	MotorRunning			: ARRAY[1..6] OF BOOL;
	
	AutoMode				: BOOL;
	
	VibrationSensorX		: ARRAY[1..6] OF REAL;
	VibrationSensorY		: ARRAY[1..6] OF REAL;
	VibrationSensorZ 		: ARRAY[1..6] OF REAL;
	VibrationSensorsEnable	: BOOL := TRUE;
	
	AirFlowRate				: REAL;
	AirPressure				: REAL;
	AirTemperature			: REAL;
	
	AirValve				: ARRAY[1..6] OF AirValveSimSignals;
	AirValveEnable			: ARRAY[1..6] OF BOOL := [TRUE, TRUE, TRUE, TRUE];
	AirValvePositionSim		: ARRAY [1..6] OF INT;
	
	ProductPosition			: INT;
	SensorProductActive		: BOOL;	
	OkProductCount			: UINT;
	NokProductCount			: UINT;	
	OkPartsPerMinRate		: UINT;	
	OkPartsPerMinHistorical	: ARRAY [1..5] OF INT;
	
	ElCurrentL1				: ARRAY[1..2] OF REAL;
	ElCurrentL2				: ARRAY[1..2] OF REAL;
	ElCurrentL3				: ARRAY[1..2] OF REAL;
	
	AmbientTemperature		: REAL;
	AmbientHumidity			: REAL;
	
	OilDiffPressure			: REAL;
	
END_VAR

// ---- POUs/PRG_10ms/PRG_01_MAIN.TcPOU
PROGRAM PRG_01_MAIN
VAR
			tonRecycle100ms			:	TON;
			tonRecycle5sec			:	TON;
END_VAR

PRG_02_DataMapping();

Simulation();

PRG_03_VibrationAnalytics();
PRG_04_AirValveAnalytics();
PRG_05_ElectricalAnalytics();
PRG_06_ElectricalMonitoring();
PRG_07_LineState();
PRG_08_ProductionStatistics();
PRG_09_PlcDiagnostic();


tonRecycle5sec(IN:=NOT tonRecycle5sec.Q, PT:=T#5S);
tonRecycle100ms(IN:=NOT tonRecycle100ms.Q, PT:=T#500MS);

// 500 ms cycle monitoring
IF tonRecycle100ms.Q THEN
	PRG_11_AirFlowAnalytics();
	
END_IF

// slow process values monitoring
IF tonRecycle5sec.Q THEN
	PRG_10_TempHumidAnalytics();
	PRG_12_OilContaminationAnalytics();
END_IF

END_PROGRAM

// ---- POUs/PRG_10ms/PRG_02_DataMapping.TcPOU
PROGRAM PRG_02_DataMapping
VAR

END_VAR


// ************** IO-Link node 1 ***************
GVL_SW.VibSensor1AccelRmsX 	:= GVL_HW.IoLinkNode1Ch1_VibAccelRmsX;
GVL_SW.VibSensor1AccelRmsY 	:= GVL_HW.IoLinkNode1Ch1_VibAccelRmsY;
GVL_SW.VibSensor1AccelRmsZ 	:= GVL_HW.IoLinkNode1Ch1_VibAccelRmsZ;
GVL_SW.VibSensor1Temp 		:= GVL_HW.IoLinkNode1Ch1_SensorTemp;

GVL_SW.VibSensor2AccelRmsX 	:= GVL_HW.IoLinkNode1Ch2_VibAccelRmsX;
GVL_SW.VibSensor2AccelRmsY 	:= GVL_HW.IoLinkNode1Ch2_VibAccelRmsY;
GVL_SW.VibSensor2AccelRmsZ 	:= GVL_HW.IoLinkNode1Ch2_VibAccelRmsZ;
GVL_SW.VibSensor2Temp 		:= GVL_HW.IoLinkNode1Ch2_SensorTemp;

GVL_SW.VibSensor3AccelRmsX 	:= GVL_HW.IoLinkNode1Ch3_VibAccelRmsX;
GVL_SW.VibSensor3AccelRmsY 	:= GVL_HW.IoLinkNode1Ch3_VibAccelRmsY;
GVL_SW.VibSensor3AccelRmsZ 	:= GVL_HW.IoLinkNode1Ch3_VibAccelRmsZ;
GVL_SW.VibSensor3Temp 		:= GVL_HW.IoLinkNode1Ch3_SensorTemp;

GVL_SW.VibSensor4AccelRmsX 	:= GVL_HW.IoLinkNode1Ch4_VibAccelRmsX;
GVL_SW.VibSensor4AccelRmsY 	:= GVL_HW.IoLinkNode1Ch4_VibAccelRmsY;
GVL_SW.VibSensor4AccelRmsZ 	:= GVL_HW.IoLinkNode1Ch4_VibAccelRmsZ;
GVL_SW.VibSensor4Temp 		:= GVL_HW.IoLinkNode1Ch4_SensorTemp;

GVL_SW.VibSensor5AccelRmsX 	:= GVL_HW.IoLinkNode1Ch5_VibAccelRmsX;
GVL_SW.VibSensor5AccelRmsY 	:= GVL_HW.IoLinkNode1Ch5_VibAccelRmsY;
GVL_SW.VibSensor5AccelRmsZ 	:= GVL_HW.IoLinkNode1Ch5_VibAccelRmsZ;
GVL_SW.VibSensor5Temp 		:= GVL_HW.IoLinkNode1Ch5_SensorTemp;

GVL_SW.VibSensor6AccelRmsX 	:= GVL_HW.IoLinkNode1Ch6_VibAccelRmsX;
GVL_SW.VibSensor6AccelRmsY 	:= GVL_HW.IoLinkNode1Ch6_VibAccelRmsY;
GVL_SW.VibSensor6AccelRmsZ 	:= GVL_HW.IoLinkNode1Ch6_VibAccelRmsZ;
GVL_SW.VibSensor6Temp 		:= GVL_HW.IoLinkNode1Ch6_SensorTemp;


// ************** IO-Link node 2 ***************
GVL_SW.AirMassFlowRate		:= GVL_HW.IoLinkNode2Ch1_MassFlowRate;	
GVL_SW.AirFlowVelocity		:= GVL_HW.IoLinkNode2Ch1_FlowVelocity;
GVL_SW.AirVolume			:= GVL_HW.IoLinkNode2Ch1_Volume;
GVL_SW.AirVolumetricFlowRate := (GVL_HW.IoLinkNode2Ch1_VolFlowRate * 1000) / 60.0;		// convert [m3/h] to [l/min]
GVL_SW.AirMass				:= GVL_HW.IoLinkNode2Ch1_Mass;
GVL_SW.AirEnergy			:= GVL_HW.IoLinkNode2Ch1_Energy;
GVL_SW.AirTemperature		:= GVL_HW.IoLinkNode2Ch1_Temperature;
GVL_SW.AirPressure			:= GVL_HW.IoLinkNode2Ch1_Pressure;

GVL_SW.AmbientTempSensor 	:=  UINT_TO_REAL( SHL(GVL_HW.IoLinkNode2Ch2_Temperature[1], 8) +  
												GVL_HW.IoLinkNode2Ch2_Temperature[2]) / 10.0;
												
GVL_SW.AmbientHumiditySensor :=  UINT_TO_REAL(SHL(GVL_HW.IoLinkNode2Ch2_Humidity[1], 8) + 
													GVL_HW.IoLinkNode2Ch2_Humidity[1] ) / 10.0;
													
													
GVL_SW.LevelSensor			:=	TO_REAL(GVL_HW.IoLinkNode2Ch3_Level) / 1000.0;			// convert to m with 1mm resolution
GVL_SW.DiffPressSensor		:= 	TO_REAL(GVL_HW.IoLinkNode2Ch4_DiffPress) / 10;			// convert to bar with 0.1 bar resolution

// Profinet IO-device data
GVL_SW.PnIoDevice_32Word_In 	:= GVL_HW.PnIoDevice_32Word_In;
GVL_SW.PnIoDevice_32DWord_In 	:= GVL_HW.PnIoDevice_32DWord_In;
GVL_SW.PnIoDevice_10Real_In		:= GVL_HW.PnIoDevice_10Real_In;
GVL_SW.PnIoDevice_10Real_Out	:= GVL_HW.PnIoDevice_10Real_Out;

// Here it's place for specified mapping of GVL_SW.PnIoDevice e.g.
// GVL_SW.Motor1.SignalStart :=  GVL_HW.PnIoDevice_32Word_In[1].0;
// GVL_SW.AnalogValue1 := GVL_HW.PnIoDevice_10Real_In[0].1;

END_PROGRAM

// ---- POUs/PRG_10ms/Simulation.TcPOU
PROGRAM Simulation
VAR
	idx			: BYTE;
	tp1Motor 	: ARRAY[1..6] OF TP;
	tp2Motor 	: ARRAY[1..6] OF TP;
	
	VibSensorBase : ARRAY[1..6] OF REAL := [0.7, 0.2, 0.3, 0.8, 0.5, 0.1];
	VibSensorOffset : ARRAY[1..6] OF REAL;
	
	AirFlowRateBase			:	REAL := 30.0;
	AirPressureBase			:	REAL := 6.0;
	AirTemperatureBase		:	REAL := 20.0;
	
	AirValve				:	ARRAY [1..6] OF Valve_Signal_Sim;
	AirValvePositionSim		: 	ARRAY [1..6] OF INT;
	
	tonProductPos			:	TON;
	rtrigProductSensor		: 	R_TRIG;
	
	tp1AutoMode				:	TP;
	tp2AutoMode				:	TP;
	tp1AutoModeTime			:	TIME := T#5S;
	tp2AutoModeTime			:	TIME := T#2S;
	rtrigAutoMode			:	R_TRIG;

	rndTime1				: INT;
	rndTime2				: INT;
	
	ElecSample1				: INT;
	ElecSample2				: INT;
	ElecCurrentOffsetL1		: REAL;
	ElecCurrentOffsetL2		: REAL;	
	ElecCurrentOffsetL3		: REAL;
	ElCurrentL1Base			: ARRAY[1..2] OF ARRAY[1..100] OF REAL := 
								[
								[0, 0, 0.1, 0.3, 0.45, 0.60, 0.70, 0.80, 0.95, 1.1, 1.3, 1.4, 1.55, 1.6, 1.59,1.55, 
								1.45, 1.3, 1.2, 1.1, 1.05, 1.0, 0.95, 0.9, 0.85, 0.83, 0.80, 0.78, 0.75, 0.74, 0.72,
								0.70, 0.69, 0.69, 0.69, 0.68, 0.68, 0.67, 0.67, 0.65, 0.64, 0.62, 0.60, 0.58, 0.58, 0.57, 0.56, 0.55, 0.55,
								0, 0, 0, 0, 0, 0, 0, 0, 0, 0],
								[0, 0, 0.1, 0.2, 0.3, 0.55, 1.0, 1.3, 1.5, 1.7, 1.8, 1.81, 1.7, 1.5, 1.2, 1.22, 1.19, 1.23,
								1.19, 1.21, 1.18, 1.22, 1.19, 1.23, 1.17, 1.21, 1.20, 1.18, 1.21, 1.18, 1.22, 1.17, 1.23,
								1.19, 1.21, 1.19, 1.20, 1.19, 1.20, 1.19, 1.21, 1.20, 1.20, 1.22, 1.19, 1.21, 1.18, 1.21, 1.2, 1.2,
								1.21, 1.20, 1.20, 1.22, 1.19, 1.21, 1.18, 1.21, 1.2, 1.2, 40(1.2)]];
								
	ElCurrentL2Base			: ARRAY[1..2] OF ARRAY[1..100] OF REAL := 
								[
								[0, 0, 0.1, 0.3, 0.45, 0.60, 0.70, 0.80, 0.95, 1.1, 1.3, 1.4, 1.55, 1.6, 1.59,1.55, 
								1.45, 1.3, 1.2, 1.1, 1.05, 1.0, 0.95, 0.9, 0.85, 0.83, 0.80, 0.78, 0.75, 0.74, 0.72,
								0.70, 0.69, 0.69, 0.69, 0.68, 0.68, 0.67, 0.67, 0.65, 0.64, 0.62, 0.60, 0.58, 0.58, 0.57, 0.56, 0.55, 0.55,
								0, 0, 0, 0, 0, 0, 0, 0, 0, 0],
								[0, 0, 0.1, 0.2, 0.3, 0.55, 1.0, 1.3, 1.5, 1.7, 1.8, 1.81, 1.7, 1.5, 1.2, 1.22, 1.19, 1.23,
								1.19, 1.21, 1.18, 1.22, 1.19, 1.23, 1.17, 1.21, 1.20, 1.18, 1.21, 1.18, 1.22, 1.17, 1.23,
								1.19, 1.21, 1.19, 1.20, 1.19, 1.20, 1.19, 1.21, 1.20, 1.20, 1.22, 1.19, 1.21, 1.18, 1.21, 1.2, 1.2,
								1.21, 1.20, 1.20, 1.22, 1.19, 1.21, 1.18, 1.21, 1.2, 1.2]];

	ElCurrentL3Base			: ARRAY[1..2] OF ARRAY[1..100] OF REAL := 
								[
								[0, 0, 0.1, 0.3, 0.45, 0.60, 0.70, 0.80, 0.95, 1.1, 1.3, 1.4, 1.55, 1.6, 1.59,1.55, 
								1.45, 1.3, 1.2, 1.1, 1.05, 1.0, 0.95, 0.9, 0.85, 0.83, 0.80, 0.78, 0.75, 0.74, 0.72,
								0.70, 0.69, 0.69, 0.69, 0.68, 0.68, 0.67, 0.67, 0.65, 0.64, 0.62, 0.60, 0.58, 0.58, 0.57, 0.56, 0.55, 0.55,
								0, 0, 0, 0, 0, 0, 0, 0, 0, 0],
								[0, 0, 0.1, 0.2, 0.3, 0.55, 1.0, 1.3, 1.5, 1.7, 1.8, 1.81, 1.7, 1.5, 1.2, 1.22, 1.19, 1.23,
								1.19, 1.21, 1.18, 1.22, 1.19, 1.23, 1.17, 1.21, 1.20, 1.18, 1.21, 1.18, 1.22, 1.17, 1.23,
								1.19, 1.21, 1.19, 1.20, 1.19, 1.20, 1.19, 1.21, 1.20, 1.20, 1.22, 1.19, 1.21, 1.18, 1.21, 1.2, 1.2,
								1.21, 1.20, 1.20, 1.22, 1.19, 1.21, 1.18, 1.21, 1.2, 1.2]];
END_VAR

IF GVL_Visu.ButtonStart THEN
	
	GVL_Visu.LineRunning := TRUE;
	// simulate motor running signals
	tp1Motor[1](IN:= NOT tp2Motor[1].Q, PT:= T#1S);
	tp2Motor[1](IN:= NOT tp1Motor[1].Q, PT:= T#500MS);
	
	tp1Motor[2](IN:= NOT tp2Motor[2].Q, PT:= T#2S);
	tp2Motor[2](IN:= NOT tp1Motor[2].Q, PT:= T#300MS);
	
	tp1Motor[3](IN:= NOT tp2Motor[3].Q, PT:= T#1.7S);
	tp2Motor[3](IN:= NOT tp1Motor[3].Q, PT:= T#500MS);
	
	tp1Motor[4](IN:= NOT tp2Motor[4].Q, PT:= T#1S);
	tp2Motor[4](IN:= NOT tp1Motor[4].Q, PT:= T#1S);
	
	tp1Motor[5](IN:= NOT tp2Motor[5].Q, PT:= T#500MS);
	tp2Motor[5](IN:= NOT tp1Motor[5].Q, PT:= T#2S);
	
	tp1Motor[6](IN:= NOT tp2Motor[6].Q, PT:= T#1S);
	tp2Motor[6](IN:= NOT tp1Motor[6].Q, PT:= T#300MS);
	
	// simulate auto/manual mode
	tp1AutoMode(IN:= NOT tp2AutoMode.Q, PT:= tp1AutoModeTime);
	tp2AutoMode(IN:= NOT tp1AutoMode.Q, PT:= tp2AutoModeTime);
	
	rtrigAutoMode(CLK:=tp1AutoMode.Q);
	
	// generate random time windows of auto and manual period  
	IF  rtrigAutoMode.Q THEN
		rndTime1 := RDM2(last:=2, low:=0, high:=70);
		tp1AutoModeTime:=T#5S + INT_TO_TIME(rndTime1*100);
		
		rndTime2 := RDM2(last:=5, low:=0, high:=30);
		tp2AutoModeTime:=T#2S + INT_TO_TIME(rndTime2*100);
	END_IF

	GVL_Visu.AutoMode := tp2AutoMode.Q;
	
	
	// simulate vibration sensors
	FOR idx := 1 TO 6 DO
		GVL_Visu.MotorRunning[idx] := tp1Motor[idx].Q;
		
		GVL_Visu.VibrationSensorX[idx] := VibSensorBase[idx] + RDM(0.4);
		GVL_Visu.VibrationSensorY[idx] := VibSensorBase[idx] + RDM(0.2);
		GVL_Visu.VibrationSensorZ[idx] := VibSensorBase[idx] + RDM(0.8);	
	END_FOR
	
	// simulate air supply sensors
	GVL_Visu.AirFlowRate 		:= AirFlowRateBase + 2* RDM(0.5);
	GVL_Visu.AirPressure		:= AirPressureBase + 2 * RDM(0.9); 
	GVL_Visu.AirTemperature		:= AirTemperatureBase + RDM(0.3);
	
	// simulate air valves
	AirValve[1](StartSim			:= TRUE, 
			    ExtendCmdTime		:= T#500MS,
			    ExtendTime 			:= T#1800MS,
			    RetractCmdTime 		:= T#600MS,
			    RetractTime  		:= T#2000MS);
			  
	AirValve[2](StartSim			:= TRUE, 
			    ExtendCmdTime		:= T#50MS,
			    ExtendTime 			:= T#180MS,
			    RetractCmdTime 		:= T#50MS,
			    RetractTime  		:= T#145MS);
				
	AirValve[3](StartSim			:= TRUE, 
			    ExtendCmdTime		:= T#100MS,
			    ExtendTime 			:= T#1200MS,
			    RetractCmdTime 		:= T#120MS,
			    RetractTime  		:= T#1500MS);
				
	AirValve[4](StartSim			:= TRUE, 
			    ExtendCmdTime		:= T#30MS,
			    ExtendTime 			:= T#120MS,
			    RetractCmdTime 		:= T#30MS,
			    RetractTime  		:= T#120MS);
				
	FOR idx := 1 TO 4 DO
		GVL_Visu.AirValve[idx].ExtendCmd := AirValve[idx].ExtendCmd;
		GVL_Visu.AirValve[idx].ExtendFeedback := AirValve[idx].ExtendFeedback;
		GVL_Visu.AirValve[idx].RetractCmd := AirValve[idx].RetractCmd;
		GVL_Visu.AirValve[idx].RetractFeedback := AirValve[idx].RetractFeedback;
		GVL_Visu.AirValvePositionSim[idx] := SEL (NOT GVL_Visu.AirValveEnable[idx], AirValve[idx].nState, 0);
	END_FOR
	
	// simulate product position on the conveyor
	tonProductPos(IN:= NOT tonProductPos.Q, PT:=T#200MS);
	IF tonProductPos.Q THEN
		GVL_Visu.ProductPosition := GVL_Visu.ProductPosition + TO_INT(GVL_Visu.LineSpeed / 5);
	END_IF
	
	IF GVL_Visu.ProductPosition >= 190 THEN
		GVL_Visu.ProductPosition := 0;
	END_IF
	
	// simulate product sensor acitivation
	IF GVL_Visu.ProductPosition >= 175 AND
		 GVL_Visu.ProductPosition <190 THEN
	GVL_Visu.SensorProductActive := TRUE;
	ELSE
		GVL_Visu.SensorProductActive := FALSE;
	END_IF;
	
	// simulate product counting
	rtrigProductSensor(CLK:=GVL_Visu.SensorProductActive);
	IF rtrigProductSensor.Q THEN
		GVL_Visu.OkProductCount := GVL_Visu.OkProductCount + 1;
	END_IF
	
	// simulate electrical current curve of motor 1
	IF GVL_Visu.MotorRunning[1] THEN
		ElecSample1 := ElecSample1+1;
		ElecSample1 := SEL(ElecSample1=60, ElecSample1, 1);
		IF ElecSample1 < 20 OR ElecSample1 > 40 THEN
			ElecCurrentOffsetL1 := RDM(0.67) * 0.05;
			ElecCurrentOffsetL2 := RDM(0.23) * 0.05;
			ElecCurrentOffsetL3 := RDM(0.72) * 0.05;
		ELSE
			ElecCurrentOffsetL1 := RDM(0.31) * 0.05;
			ElecCurrentOffsetL2 := RDM(0.63) * 0.05;
			ElecCurrentOffsetL3 := RDM(0.46) * 0.05;
		END_IF
		GVL_Visu.ElCurrentL1[1] := 	ElCurrentL1Base[1][ElecSample1];
		GVL_Visu.ElCurrentL2[1] := 	ElCurrentL1Base[1][ElecSample1];
		GVL_Visu.ElCurrentL3[1] := 	ElCurrentL1Base[1][ElecSample1];
	ELSE
		ElecSample1 := 0;
		GVL_Visu.ElCurrentL1[1] := 0;
		GVL_Visu.ElCurrentL2[1] := 0;
		GVL_Visu.ElCurrentL3[1] := 0;
	END_IF
	
	// simulate electrical current curve of motor 2
	IF GVL_Visu.MotorRunning[2] THEN
		ElecSample2 := ElecSample2+1;
		ElecSample2 := SEL(ElecSample2=60, ElecSample2, 1);
		GVL_Visu.ElCurrentL1[2] := 	ElCurrentL1Base[2][ElecSample2];
		GVL_Visu.ElCurrentL2[2] := 	ElCurrentL2Base[2][ElecSample2];
		GVL_Visu.ElCurrentL3[2] := 	ElCurrentL3Base[2][ElecSample2];
	ELSE
		ElecSample2 := 0;
		GVL_Visu.ElCurrentL1[2] := 0;
		GVL_Visu.ElCurrentL2[2] := 0;
		GVL_Visu.ElCurrentL3[2] := 0;
	END_IF
	
	// simulate ambient temperature & humidity
	GVL_Visu.AmbientTemperature := 19.0 + 2* RDM(0.7);
	GVL_Visu.AmbientHumidity	:= 60.0 + 3 * RDM(0.5);
	
	// simulate pressure difference for oil contamination sensor
	GVL_Visu.OilDiffPressure := 0.22 + RDM(0.1) * 0.2;
  

ELSE
	GVL_Visu.LineRunning := FALSE;
	tp1AutoMode(IN:=FALSE);
	tp2AutoMode(IN:=FALSE);
	
	GVL_Visu.AutoMode := tp1AutoMode.Q;
	
	FOR idx := 1 TO 4 DO
		AirValve[idx](StartSim := FALSE);
	END_FOR
	
	FOR idx := 1 TO 6 DO
		tp1Motor[idx](IN:= FALSE);
		tp2Motor[idx](IN:= FALSE);	
		GVL_Visu.MotorRunning[idx] := tp1Motor[idx].Q;		
	END_FOR
	
	GVL_Visu.ElCurrentL1[1] := 0;
	GVL_Visu.ElCurrentL2[1] := 0;
	GVL_Visu.ElCurrentL3[1] := 0;
	
	GVL_Visu.ElCurrentL1[2] := 0;
	GVL_Visu.ElCurrentL2[2] := 0;
	GVL_Visu.ElCurrentL3[2] := 0;
	
END_IF

END_PROGRAM

// ---- POUs/FB/Generic/Valve_Signal_Sim.TcPOU
FUNCTION_BLOCK Valve_Signal_Sim
VAR_INPUT
	StartSim : BOOL;
	
	ExtendCmdTime	:	TIME;
	ExtendTime		:	TIME;
	RetractCmdTime	:	TIME;
	RetractTime		:	TIME;
END_VAR
VAR_OUTPUT
	ExtendCmd 		: 	BOOL;
	ExtendFeedback 	: 	BOOL;
	RetractCmd 		: 	BOOL;
	RetractFeedback : 	BOOL;
	SequenceStatus 	: 	INT;
	
END_VAR
VAR
	tonExtendCmd	: TON;
	tonExtend		: TON;
	tonRetractCmd	: TON;
	tonRetract		: TON;
	
	ExtendPos_ton: TON; //czas przebywania na pozycji Extend
	RetractPos_ton: TON; //czas przebywania na pozycji Retract
	
	nState : INT;
	
	// sequence watchdog
	tonWatchdog		: TON;
	rtrigStartSim	: R_TRIG;

	Step20Cnt: INT;
	Step30Cnt: INT;
END_VAR

rtrigStartSim(CLK:=StartSim);

CASE nState OF
0:
	SequenceStatus := 0;
	tonExtendCmd.IN := FALSE;
	tonExtend.IN := FALSE;
	tonRetractCmd.IN := FALSE;
	tonRetract.IN := FALSE;
	
	RetractFeedback := TRUE;
	
	IF rtrigStartSim.Q THEN
		nState := nState + 10;
		tonWatchdog.IN := TRUE;
	END_IF

10:
	SequenceStatus := 10;
	ExtendCmd := TRUE;
	tonExtendCmd.IN := TRUE;
	IF tonExtendCmd.Q THEN
		nState := nState + 10;
		tonExtendCmd.IN := FALSE;
	END_IF
20:	
	SequenceStatus := 20;
	RetractFeedback :=FALSE;
	tonExtend.IN := TRUE;
	IF tonExtend.Q THEN
		nState := nState + 10;
		tonExtend.IN := FALSE;
	END_IF
		
	
30:
	SequenceStatus := 30;
	ExtendFeedback := TRUE;
	ExtendCmd := FALSE;
	ExtendPos_ton.IN := TRUE;
	IF ExtendPos_ton.Q THEN
		nState := nState + 10;
		ExtendPos_ton.IN := FALSE;
	END_IF


40:
	SequenceStatus := 40;
	RetractCmd := TRUE;
	tonRetractCmd.IN := TRUE;
	IF tonRetractCmd.Q THEN
		nState := nState + 10;
		tonRetractCmd.IN := FALSE;
	END_IF
50:
	SequenceStatus := 50;
	ExtendFeedback :=FALSE;
	tonRetract.IN := TRUE;
	IF tonRetract.Q THEN
		nState := nState + 10;
		tonRetract.IN := FALSE;
	END_IF
60:
	SequenceStatus := 60;
	RetractFeedback := TRUE;
	RetractCmd := FALSE;
	RetractPos_ton.IN := TRUE;
	IF RetractPos_ton.Q THEN
		nState := 10;
		RetractPos_ton.IN := FALSE;
	END_IF

	
END_CASE

IF StartSim = FALSE THEN
	nState := 0;
END_IF

tonExtendCmd(PT:=ExtendCmdTime);
tonExtend(PT:=ExtendTime);
tonRetractCmd(PT:=RetractCmdTime);
tonRetract(PT:=RetractTime);

ExtendPos_ton(PT:=T#500MS);
RetractPos_ton(PT:=T#500MS);
tonWatchdog(PT:=T#2H);

END_FUNCTION_BLOCK

// ---- POUs/PRG_10ms/PRG_03_VibrationAnalytics.TcPOU
PROGRAM PRG_03_VibrationAnalytics
VAR
	VibSensor					: ARRAY [1..6] OF VibrationSensor;
	
	
	{attribute 'OPC.UA.DA' := '0'}
	{attribute 'OPC.UA.DA.Access' := '1'}			// read only
	{attribute 'OPC.UA.DA.StructuredType' := '1'}
	VibSensorStruct01			: VibAccelarationDataModel;
	
	{attribute 'OPC.UA.DA' := '0'}
	{attribute 'OPC.UA.DA.Access' := '1'}			// read only
	{attribute 'OPC.UA.DA.StructuredType' := '1'}
	VibSensorStruct02			: VibAccelarationDataModel;

	{attribute 'OPC.UA.DA' := '0'}
	{attribute 'OPC.UA.DA.Access' := '1'}			// read only
	{attribute 'OPC.UA.DA.StructuredType' := '1'}
	VibSensorStruct03			: VibAccelarationDataModel;
	
	{attribute 'OPC.UA.DA' := '0'}
	{attribute 'OPC.UA.DA.Access' := '1'}			// read only
	{attribute 'OPC.UA.DA.StructuredType' := '1'}
	VibSensorStruct04			: VibAccelarationDataModel;
	
	{attribute 'OPC.UA.DA' := '0'}
	{attribute 'OPC.UA.DA.Access' := '1'}			// read only
	{attribute 'OPC.UA.DA.StructuredType' := '1'}
	VibSensorStruct05			: VibAccelarationDataModel;
	
	{attribute 'OPC.UA.DA' := '0'}
	{attribute 'OPC.UA.DA.Access' := '1'}			// read only
	{attribute 'OPC.UA.DA.StructuredType' := '1'}
	VibSensorStruct06			: VibAccelarationDataModel;
	

END_VAR


// PAGE Vibration Sensor 1 ----
VibSensor[1](
    LineName := GVL_const.LineName,
    MachineName := GVL_const.MachineName,
    SensorName := GVL_const.VibSensor1,
    TimeStamp := GVL_SW.Unix_TimeStamp,
    VibAccelX := GVL_Visu.VibrationSensorX[1],
    VibAccelY := GVL_Visu.VibrationSensorY[1],
    VibAccelZ := GVL_Visu.VibrationSensorZ[1],
    SensorTemperature := GVL_SW.VibSensor1Temp,
    MotorState := GVL_Visu.MotorRunning[1],
    Enable := GVL_Visu.LineRunning AND GVL_Visu.VibrationSensorsEnable); // VibrationSensor
VibSensorStruct01 := VibSensor[1].OpcUaVal;

// PAGE Vibration Sensor 2 ---
VibSensor[2](
    LineName := GVL_const.LineName,
    MachineName := GVL_const.MachineName,
    SensorName := GVL_const.VibSensor2,
    TimeStamp := GVL_SW.Unix_TimeStamp,
    VibAccelX := GVL_Visu.VibrationSensorX[2],
    VibAccelY := GVL_Visu.VibrationSensorY[2],
    VibAccelZ := GVL_Visu.VibrationSensorZ[2],
    SensorTemperature := GVL_SW.VibSensor2Temp,
    MotorState := GVL_Visu.MotorRunning[2],
    Enable := GVL_Visu.LineRunning AND GVL_Visu.VibrationSensorsEnable); // VibrationSensor
VibSensorStruct02 := VibSensor[2].OpcUaVal;

// PAGE Vibration Sensor 3 ---
VibSensor[3](
    LineName := GVL_const.LineName,
    MachineName := GVL_const.MachineName,
    SensorName := GVL_const.VibSensor3,
    TimeStamp := GVL_SW.Unix_TimeStamp,
    VibAccelX := GVL_Visu.VibrationSensorX[3],
    VibAccelY := GVL_Visu.VibrationSensorY[3],
    VibAccelZ := GVL_Visu.VibrationSensorZ[3],
    SensorTemperature := GVL_SW.VibSensor3Temp,
    MotorState := GVL_Visu.MotorRunning[3],
    Enable := GVL_Visu.LineRunning AND GVL_Visu.VibrationSensorsEnable); // VibrationSensor
VibSensorStruct03 := VibSensor[3].OpcUaVal;

// PAGE Vibration Sensor 4 ---
VibSensor[4](
    LineName := GVL_const.LineName,
    MachineName := GVL_const.MachineName,
    SensorName := GVL_const.VibSensor4,
    TimeStamp := GVL_SW.Unix_TimeStamp,
    VibAccelX := GVL_Visu.VibrationSensorX[4],
    VibAccelY := GVL_Visu.VibrationSensorY[4],
    VibAccelZ := GVL_Visu.VibrationSensorZ[4],
    SensorTemperature := GVL_SW.VibSensor4Temp,
    MotorState := GVL_Visu.MotorRunning[4],
    Enable := GVL_Visu.LineRunning AND GVL_Visu.VibrationSensorsEnable); // VibrationSensor
VibSensorStruct04 := VibSensor[4].OpcUaVal;

// PAGE Vibration Sensor 5 ---
VibSensor[5](
    LineName := GVL_const.LineName,
    MachineName := GVL_const.MachineName,
    SensorName := GVL_const.VibSensor5,
    TimeStamp := GVL_SW.Unix_TimeStamp,
    VibAccelX := GVL_Visu.VibrationSensorX[5],
    VibAccelY := GVL_Visu.VibrationSensorY[5],
    VibAccelZ := GVL_Visu.VibrationSensorZ[5],
    SensorTemperature := GVL_SW.VibSensor5Temp,
    MotorState := GVL_Visu.MotorRunning[5],
    Enable := GVL_Visu.LineRunning AND GVL_Visu.VibrationSensorsEnable); // VibrationSensor
VibSensorStruct05 := VibSensor[5].OpcUaVal;

// PAGE Vibration Sensor 6 ---
VibSensor[6](
    LineName := GVL_const.LineName,
    MachineName := GVL_const.MachineName,
    SensorName := GVL_const.VibSensor6,
    TimeStamp := GVL_SW.Unix_TimeStamp,
    VibAccelX := GVL_Visu.VibrationSensorX[6],
    VibAccelY := GVL_Visu.VibrationSensorY[6],
    VibAccelZ := GVL_Visu.VibrationSensorZ[6],
    SensorTemperature := GVL_SW.VibSensor6Temp,
    MotorState := GVL_Visu.MotorRunning[6],
    Enable := GVL_Visu.LineRunning AND GVL_Visu.VibrationSensorsEnable); // VibrationSensor
VibSensorStruct06 := VibSensor[6].OpcUaVal;
// GVL.BS1_Accel_RMS_X: input not connected
// GVL.BS1_Accel_RMS_Y: input not connected
// GVL.BS1_Accel_RMS_Z: input not connected
// GVL.Drv_RotTable_25N0_M10_RUNNING: input not connected
// GVL.AutoMode: input not connected
// GVL.BS2_Accel_RMS_X: input not connected
// GVL.BS2_Accel_RMS_Y: input not connected
// GVL.BS2_Accel_RMS_Z: input not connected
// GVL.Drv_RotTable_25N0_M10_RUNNING: input not connected
// GVL.AutoMode: input not connected
// GVL.BS3_Accel_RMS_X: input not connected
// GVL.BS3_Accel_RMS_Y: input not connected
// GVL.BS3_Accel_RMS_Z: input not connected
// GVL.Drv_RotTable_25N0_M10_RUNNING: input not connected
// GVL.AutoMode: input not connected
// GVL.BS4_Accel_RMS_X: input not connected
// GVL.BS4_Accel_RMS_Y: input not connected
// GVL.BS4_Accel_RMS_Z: input not connected
// GVL.Drv_RotTable_25N0_M10_RUNNING: input not connected
// GVL.AutoMode: input not connected
// GVL.BS5_Accel_RMS_X: input not connected
// GVL.BS5_Accel_RMS_Y: input not connected
// GVL.BS5_Accel_RMS_Z: input not connected
// GVL.Drv_InfeedBelt2_10N31_M21_RIGHT_RUNNING: input not connected
// GVL.AutoMode: input not connected
// GVL.BS6_Accel_RMS_X: input not connected
// GVL.BS6_Accel_RMS_Y: input not connected
// GVL.BS6_Accel_RMS_Z: input not connected
// GVL.Drv_InfeedBelt2_10N31_M21_RIGHT_RUNNING: input not connected
// GVL.AutoMode: input not connected

END_PROGRAM

// ---- POUs/FB/OPC_UA/VibrationSensor.TcPOU
FUNCTION_BLOCK VibrationSensor
VAR_INPUT
	LineName			: STRING(40);
	MachineName 		: STRING(40);
	SensorName			: STRING(40);
	TimeStamp			: ULINT;
	VibAccelX			: REAL;
    VibAccelY			: REAL;
    VibAccelZ			: REAL;	
    SensorTemperature	: REAL;
	MotorState			: BOOL;	
	Enable				: BOOL;
END_VAR
VAR_OUTPUT
	OpcUaVal			: VibAccelarationDataModel;
END_VAR
VAR
	SetParameter 		: BOOL := TRUE;
	
	// state machine
	nState				: INT := 0;
	
	stValues			: VibAccelarationDataModel;	

	// motor status 
	rtrigMotorState		: R_TRIG;
	ftrigMotorState		: F_TRIG;
	 
	// safety watchdog
	tonWatchdog 		: TON;
	
	StoppingCntr 		: INT;
	StoppedCntr 		: INT;
	
	 //Motor state
	 StartingState		: BOOL := FALSE;
     RunningState		: BOOL := FALSE;
     StoppingState		: BOOL := FALSE;
     StoppedState		: BOOL := FALSE;
	 DriveStates		: DriveState_DataModel; 
	
END_VAR

(*
This FB calculates analytics when motor status is TRUE.
During this state vibration's values from axis x,y,z from the sensor
are accumulated and will create output struct for OPC UA  at falling
edge of the motor state.
Vibration sensor needs to be located ar the motor or its gearing/coupling 
*)

IF SetParameter THEN
	SetParameter := FALSE;
	
	// constant entry in struct
	stValues.LineName := LineName;
	stValues.MachineName := MachineName;
	stValues.SensorName := SensorName;
END_IF


// detect motor state (running/stopped)
rtrigMotorState(CLK:=MotorState);
ftrigMotorState(CLK:=MotorState);

IF ENABLE THEN
	CASE nState OF
	0:
		ClearData();
		
		IF rtrigMotorState.Q THEN
			tonWatchdog.IN := TRUE;
			nState := 10;
		END_IF
		
	10:
	// RUNNING
		RunningState := TRUE;
		stValues.TimeStamp := TimeStamp;
		stValues.VibAccelTotRmsX := stValues.VibAccelTotRmsX + VibAccelX;
		stValues.VibAccelTotRmsY := stValues.VibAccelTotRmsY + VibAccelY;
		stValues.VibAccelTotRmsZ := stValues.VibAccelTotRmsZ + VibAccelZ;
		stValues.SensorTemperature := SensorTemperature;
	
		IF ftrigMotorState.Q THEN
			RunningState := FALSE;
			nState := 20;
		END_IF
	
	20:
	// STOPPING
		StoppingState := TRUE;
		stValues.TimeStamp := TimeStamp;
		stValues.VibAccelTotRmsX := stValues.VibAccelTotRmsX + VibAccelX;
		stValues.VibAccelTotRmsY := stValues.VibAccelTotRmsY + VibAccelY;
		stValues.VibAccelTotRmsZ := stValues.VibAccelTotRmsZ + VibAccelZ;
		stValues.SensorTemperature := SensorTemperature;
		
		StoppingCntr := StoppingCntr + 1;
		
		IF StoppingCntr = 2 THEN
			StoppingState := FALSE;
			nState := 30;
		END_IF
	
	30:
	// STOPPED
		StoppedState := TRUE;
		stValues.TimeStamp := TimeStamp;
		stValues.VibAccelTotRmsX := ROUND(stValues.VibAccelTotRmsX + VibAccelX, 4);
		stValues.VibAccelTotRmsY := ROUND(stValues.VibAccelTotRmsY + VibAccelY, 4);
		stValues.VibAccelTotRmsZ := ROUND(stValues.VibAccelTotRmsZ + VibAccelZ, 4);
		stValues.SensorTemperature := ROUND(SensorTemperature, 2);
	
		StoppedCntr := StoppedCntr + 1;
		
		IF StoppedCntr = 2 THEN
			StoppedState := FALSE;
			// provide measurement OPC UA data
			OpcUaVal := stValues;
			nState := 0;
		END_IF
		
		tonWatchdog.IN := FALSE;
		
	END_CASE
	
	//Watchdog 7 seconds, restart of sequence
	IF tonWatchdog.ET > T#7S AND nState <> 0 THEN
		nState := 0;
	END_IF
ELSE
	tonWatchdog.IN := FALSE;
	ClearData();
END_IF

tonWatchdog(PT:=T#10S);

METHOD ClearData
VAR_INPUT
END_VAR
nState			:= 0;
StoppingCntr 	:= 0;
StoppedCntr 	:= 0;
RunningState 	:= FALSE;
StoppingState 	:= FALSE;
StoppedState 	:= FALSE;
stValues.VibAccelTotRmsX := 0.0;
stValues.VibAccelTotRmsY := 0.0;
stValues.VibAccelTotRmsZ := 0.0;
END_METHOD

END_FUNCTION_BLOCK

// ---- POUs/PRG_1ms/TimeStamp.TcPOU
PROGRAM TimeStamp
VAR
	UnixTime: UnixTimestamp;
END_VAR

UnixTime(SyncTimeEnable := TRUE);

GVL_SW.Unix_TimeStamp := UnixTime.Milliseconds;

END_PROGRAM

// ---- POUs/FB/Generic/UnixTimestamp.TcPOU
FUNCTION_BLOCK UnixTimestamp
VAR_INPUT
	SyncTimeEnable : BOOL;
END_VAR
VAR_OUTPUT
	Seconds: ULINT;
    Milliseconds: ULINT;
	SyncTimeValid : BOOL;
END_VAR
VAR
	localSystemTime : FB_LocalSystemTime := (dwCycle := 1 );
    getTimeZoneInformation : FB_GetTimeZoneInformation;
    timeZoneInformation : ST_TimeZoneInformation;
    specificLocalTimeToFileTime : FB_TzSpecificLocalTimeToFileTime;
    fileTime: T_FILETIME;
    onZerothSecondLastCycle : BOOL;
END_VAR

// Get local system time
localSystemTime(bEnable := SyncTimeEnable);

IF(localSystemTime.bValid)THEN
	// On the zeroth second of each minutesync timezone information
	IF (timeZoneInformation.standardName = '' OR (localSystemTime.systemTime.wSecond = 0 AND NOT onZerothSecondLastCycle)) THEN
    	getTimeZoneInformation(sNetID := '', bExecute := TRUE, tzInfo => timeZoneInformation);
	END_IF;

	// Convert local system time to unix timestamps
	specificLocalTimeToFileTime(in := Tc2_Utilities.SYSTEMTIME_TO_FILETIME(localSystemTime.systemTime), tzInfo := timeZoneInformation, out => fileTime);
	//seconds := (SHL(DWORD_TO_ULINT(fileTime.dwHighDateTime), 32) + DWORD_TO_ULINT(fileTime.dwLowDateTime)) / 10000000 - 11644473600;
	milliseconds := (SHL(DWORD_TO_ULINT(fileTime.dwHighDateTime), 32) + DWORD_TO_ULINT(fileTime.dwLowDateTime)) / 10000 - 11644473600000;

	onZerothSecondLastCycle := localSystemTime.systemTime.wSecond = 0;
	SyncTimeValid := TRUE;
ELSE
	SyncTimeValid := FALSE;
END_IF

END_FUNCTION_BLOCK

// ---- POUs/PRG_10ms/PRG_04_AirValveAnalytics.TcPOU
PROGRAM PRG_04_AirValveAnalytics
VAR	
	AirValve							: ARRAY [1..6] OF Valve2Cmd2FB;
	
	{attribute 'OPC.UA.DA' := '0'}
	{attribute 'OPC.UA.DA.Access' := '1'}			// read only
	{attribute 'OPC.UA.DA.StructuredType' := '1'}
	AirValveStruct01					: ValveTravelTime_DataModel;
	
	{attribute 'OPC.UA.DA' := '0'}
	{attribute 'OPC.UA.DA.Access' := '1'}			// read only
	{attribute 'OPC.UA.DA.StructuredType' := '1'}
	AirValveStruct02					: ValveTravelTime_DataModel;
	

	AirValveStruct03						: ValveTravelTime_DataModel;
	AirValveStruct04						: ValveTravelTime_DataModel;
	

END_VAR


// PAGE Air valve 1 ---
AirValve[1](
    LineName := GVL_const.LineName,
    MachineName := GVL_const.MachineName,
    ValveName := GVL_const.AirValve1,
    ExtendCmd := GVL_Visu.AirValve[1].ExtendCmd,
    ExtendFeedback := GVL_Visu.AirValve[1].ExtendFeedback,
    RetractCmd := GVL_Visu.AirValve[1].RetractCmd,
    RetractFeedback := GVL_Visu.AirValve[1].RetractFeedback,
    TimeStamp := GVL_SW.Unix_TimeStamp,
    Enable := GVL_Visu.LineRunning AND GVL_Visu.AirValveEnable[1]); // Valve2Cmd2FB
AirValveStruct01 := AirValve[1].OpcUaVal;

// PAGE Air valve 2 ---
AirValveStruct02 := AirValve[2].OpcUaVal;
AirValve[2](
    LineName := GVL_const.LineName,
    MachineName := GVL_const.MachineName,
    ValveName := GVL_const.AirValve2,
    ExtendCmd := GVL_Visu.AirValve[2].ExtendCmd,
    ExtendFeedback := GVL_Visu.AirValve[2].ExtendFeedback,
    RetractCmd := GVL_Visu.AirValve[2].RetractCmd,
    RetractFeedback := GVL_Visu.AirValve[2].RetractFeedback,
    TimeStamp := GVL_SW.Unix_TimeStamp,
    Enable := GVL_Visu.LineRunning AND GVL_Visu.AirValveEnable[2]); // Valve2Cmd2FB

// PAGE Air valve 3 ---
AirValveStruct03 := AirValve[3].OpcUaVal;
AirValve[3](
    LineName := GVL_const.LineName,
    MachineName := GVL_const.MachineName,
    ValveName := GVL_const.AirValve3,
    ExtendCmd := GVL_Visu.AirValve[3].ExtendCmd,
    ExtendFeedback := GVL_Visu.AirValve[3].ExtendFeedback,
    RetractCmd := GVL_Visu.AirValve[3].RetractCmd,
    RetractFeedback := GVL_Visu.AirValve[3].RetractFeedback,
    TimeStamp := GVL_SW.Unix_TimeStamp,
    Enable := GVL_Visu.LineRunning AND GVL_Visu.AirValveEnable[3]); // Valve2Cmd2FB

// PAGE Air valve 4 ---
AirValveStruct04 := AirValve[4].OpcUaVal;
AirValve[4](
    LineName := GVL_const.LineName,
    MachineName := GVL_const.MachineName,
    ValveName := GVL_const.AirValve4,
    ExtendCmd := GVL_Visu.AirValve[4].ExtendCmd,
    ExtendFeedback := GVL_Visu.AirValve[4].ExtendFeedback,
    RetractCmd := GVL_Visu.AirValve[4].RetractCmd,
    RetractFeedback := GVL_Visu.AirValve[4].RetractFeedback,
    TimeStamp := GVL_SW.Unix_TimeStamp,
    Enable := GVL_Visu.LineRunning AND GVL_Visu.AirValveEnable[4]); // Valve2Cmd2FB

END_PROGRAM

// ---- POUs/FB/OPC_UA/Valve2Cmd2FB.TcPOU
FUNCTION_BLOCK Valve2Cmd2FB
VAR_INPUT
	LineName 			: STRING(40);
	MachineName 		: STRING(40);
	ValveName 			: STRING(40);
	ExtendCmd 			: BOOL;							// command EXTEND
	ExtendFeedback 		: BOOL;							// sensor feedback EXTEND
	RetractCmd 			: BOOL;							// command RETRACT
	RetractFeedback 	: BOOL;							// sensor feedback RETRACT
	MaxExtendTime		: TIME := T#7S;
	MaxRetractTime		: TIME := T#7S;
	TimeStamp 			: ULINT;
	Enable				: BOOL;
END_VAR
VAR_OUTPUT
	
	// measured travel times
	ExtendCmdTime 		: INT;			//time between Extend Command and deactivation of Home(Retract) sensor
	ExtendTime 			: INT;			//time between deactivation of Home(Retract) sensor and activation of Work(Extend) sensor
	RetractCmdTime 		: INT;			//time between Retract Command and deactivation of Work(Extend) sensor
	RetractTime 		: INT;			//time between deactivation of Work(Extend) sensor and activation od Home(retract) sensor

	OpcUaVal			: ValveTravelTime_DataModel;
END_VAR
VAR
	SetParameter : BOOL := TRUE;
	
	// enable status edge detection
	rtrigEnableStatus	: R_TRIG;
	ftrigEnableStatus	: F_TRIG;
		
	// state machine
	nExtendState			: INT;
	nRetractState			: INT;
	
	// ton for time measurement	
	tonExtendCmdTime		: TON;
	tonExtendTime			: TON;
	tonRetractCmdTime		: TON;
	tonRetractTime			: TON;
	
	// watchdog for travel time monitoring
	WatchdogExtendSequence: TON;
	WatchdogRetractSequence: TON;
	
	// temporary times
	ExtendCmdT			: TIME;
	ExtendT				: TIME;
	RetractCmdT			: TIME;
	RetractT			: TIME;
	
	// commands edge detection
	rtrigExtendCmd: R_TRIG;
	rtrigRetractCmd: R_TRIG;


	stValues		: ValveTravelTime_DataModel;
	
	// Time Types 
	TimeTypeExtendCmd 			: STRING := 'ExtendCmdTime';
	TimeTypeExtend 				: STRING := 'ExtendTime';
	TimeTypeRetractCmd 			: STRING := 'RetractCmdTime';
	TimeTypeRetract 			: STRING := 'RetractTime';
	
	// temporary mqtt topic
	TopicString : STRING;

END_VAR

(*
This FB calculates extend and retract time of
air valve based on command and feedback status.
Results are put inot OPC UA struct.
*)
IF Enable THEN		
		
		//detect edges of command
		rtrigRetractCmd(CLK:=RetractCmd);
		rtrigExtendCmd(CLK:=ExtendCmd);
		
		IF SetParameter THEN
			SetParameter := FALSE;
			
			// constant entry in json payload
			stValues.LineName 		:= LineName;
			stValues.MachineName 	:= MachineName;
			stValues.ValveName 		:= ValveName;
			stValues.TimeType		:= '';
		END_IF
		
		// evaluate analytics & sequence only when Enable = true
		IF rtrigEnableStatus.Q THEN
			nExtendState := 0;
			nRetractState := 0;
		END_IF;

		// disable analytics
		IF ftrigEnableStatus.Q THEN
			nExtendState := -1;
			nRetractState := -1;
		END_IF
				
		// valve extend sequence
		CASE nExtendState OF
		0:
			// initialization
			tonExtendCmdTime.IN  			:= FALSE;
			tonExtendTime.IN  				:= FALSE;
			WatchDogExtendSequence.IN  		:= FALSE;
		
			// extend command COMING
			IF rtrigExtendCmd.Q THEN
				tonExtendCmdTime.IN := TRUE; 		
				WatchDogExtendSequence.IN := TRUE; 	
				nExtendState := 10;
			END_IF
		10:
			nExtendState := 20;
		20:
			// Retract Feedback GONE
			IF NOT RetractFeedback THEN
				tonExtendCmdTime.IN := FALSE;
				stValues.timeStamp := TimeStamp; 		
				tonExtendTime.IN := TRUE; 			
				ExtendCmdT := tonExtendCmdTime.ET; 
				nExtendState := 30;
			END_IF
		30:
			// measure extend command time
			ExtendCmdTime := TIME_TO_INT(ExtendCmdT);
			stValues.TimeType := TimeTypeExtendCmd;
			stValues.TimeValue := ExtendCmdTime;
			
			// provide measurement OPC UA data for ExtendCmd Time
			OpcUaVal := stValues;
			
			IF ExtendCmd AND NOT RetractFeedback THEN
				nExtendState := 40;
			END_IF
		40:

			// extend feedback COMING 
			IF ExtendFeedback THEN
				tonExtendTime.IN := FALSE;
				stValues.timeStamp := TimeStamp;
				ExtendT := tonExtendTime.ET;
				nExtendState := 50;
			END_IF
		50:
			// measure extend time
			ExtendTime := TIME_TO_INT(ExtendT);
			WatchDogExtendSequence.IN:= FALSE;
			stValues.TimeType := TimeTypeExtend;
			stValues.TimeValue := ExtendTime;
			
			// provide measurement OPC UA data for Extend Time
			OpcUaVal := stValues;
			
			nExtendState := 0;
		999:
			// error handling if needed
		END_CASE
		
		// watchdog of extend sequence time. If time exceeded then restart sequence
		IF WatchDogExtendSequence.ET > MaxExtendTime THEN
			nExtendState := 0;
		END_IF
		
		
		
		// valve retract sequence
		CASE nRetractState OF
		0:
			// initialization
			tonRetractCmdTime.IN  		:= FALSE;
			tonRetractTime.IN 			:= FALSE;
			WatchDogRetractSequence.IN 	:= FALSE;
			
			// retract command COMING
			IF rtrigRetractCmd.Q THEN
				tonRetractCmdTime.IN := TRUE; 
				WatchDogRetractSequence.IN := TRUE;
				nRetractState := 10;
			END_IF
		10:
			nRetractState := 20;
		20:
			// Extend Feedback GONE
			IF NOT ExtendFeedback THEN
				tonRetractCmdTime.IN := FALSE;
				stValues.timeStamp := TimeStamp;
				tonRetractTime.IN := TRUE; 
				RetractCmdT := tonRetractCmdTime.ET;
				nRetractState := 30;	
			END_IF
		30:
			// measure retract command time
			RetractCmdTime := TIME_TO_INT(RetractCmdT);
			stValues.TimeType := TimeTypeRetractCmd;
			stValues.TimeValue := RetractCmdTime;
			
			// provide measurement OPC UA data for RetractCmd Time
			OpcUaVal := stValues;
			
			IF RetractCmd AND NOT ExtendFeedback THEN
				nRetractState := 40;	
			END_IF
		40:
			// retract feedback COMING 
			IF RetractFeedback THEN
				tonRetractTime.IN := FALSE;
				stValues.timeStamp := TimeStamp;
				RetractT := tonRetractTime.ET;
				nRetractState := 50;
			END_IF
		50:
			// measure retract time
			RetractTime := TIME_TO_INT(RetractT);
			WatchDogRetractSequence.IN:= FALSE;
			stValues.TimeType := TimeTypeRetract;
			stValues.TimeValue := RetractTime;
			
			// provide measurement OPC UA data for Retract Time
			OpcUaVal := stValues;
			
			nRetractState := 0;
		999:
			// error handling if needed 
		END_CASE
		
		// watchdog of retract sequence time. If time exceeded then restart sequence
		IF WatchDogRetractSequence.ET > MaxRetractTime THEN
			nExtendState := 0;
		END_IF
		
		tonExtendCmdTime(PT:=T#10S);
		tonExtendTime(PT:=T#10S);
		tonRetractCmdTime(PT:=T#10S);
		tonRetractTime(PT:=T#10S);
		WatchDogExtendSequence(PT:=T#10S);
		WatchDogRetractSequence(PT:=T#10S);

ELSE
;
END_IF

END_FUNCTION_BLOCK

// ---- POUs/PRG_10ms/PRG_05_ElectricalAnalytics.TcPOU
PROGRAM PRG_05_ElectricalAnalytics
VAR
	ElectricalDevice				: ARRAY[1..2] OF ElectricalDevicePeriodicOper;
	
	{attribute 'OPC.UA.DA' := '0'}					// enable/disable to OPC UA
	{attribute 'OPC.UA.DA.Access' := '1'}			// read only
	{attribute 'OPC.UA.DA.StructuredType' := '1'}	// define variable as STRUCT for OPC UA
	ElectPeriodicDeviceStruct01		: ElectrDevicePeriodicOper_DataModel;
	
	ElectPeriodicDeviceStruct02		: ElectrDevicePeriodicOper_DataModel;
		
	SyncPulseElecDevice1: TP;
	SyncPulseElecDevice2: TP;
END_VAR
VAR // added by the converter: edge detectors and wires of the graphical bodies
    _s1, _s2 : ElectrDataEthCAT;
END_VAR


// PAGE Electrical Motor1 ---
// Read electrical data from EL3443 module and send  it by MQTT during device RUN state.
// It allows analytics of periodically switched device
// compose _s1 : ElectrDataEthCAT
_s1.ActPowerTot := Main_500us.ElectricalDevice1.stVariantValues.stTotal.fPtot;
_s1.ReactPowerTot := Main_500us.ElectricalDevice1.stVariantValues.stTotal.fQtot;
_s1.ApparPowerTot := Main_500us.ElectricalDevice1.stVariantValues.stTotal.fStot;
_s1.PowerFact := Main_500us.ElectricalDevice1.stVariantValues.stTotal.fPower_Factor;
_s1.PQF := Main_500us.ElectricalDevice1.stVariantValues.stTotal.fPQF;
_s1.ActPowerL1 := Main_500us.ActPowL1ElecDevice1;
_s1.ReactPowerL1 := Main_500us.ReactPowL1ElecDevice1;
_s1.ApparPowerL1 := Main_500us.AppPowL1ElecDevice1;
_s1.CurrentL1 := GVL_Visu.ElCurrentL1[1];
_s1.VoltL1 := Main_500us.VoltL1ElecDevice1;
_s1.PowFactL1 := Main_500us.PowFactL1ElecDevice1;
_s1.VoltL1_THD := Main_500us.ElectricalDevice1.stVariantValues.astLx[1].fTHD_U;
_s1.CurrentL1_THD := Main_500us.ElectricalDevice1.stVariantValues.astLx[1].fTHD_I;
_s1.CurrentL1_harm := Main_500us.ElectricalDevice1.stVariantValues.astLx[1].fHarmonics_I;
_s1.ActPowerL2 := Main_500us.ActPowL2ElecDevice1;
_s1.ReactPowerL2 := Main_500us.ReactPowL2ElecDevice1;
_s1.ApparPowerL2 := Main_500us.AppPowL2ElecDevice1;
_s1.CurrentL2 := GVL_Visu.ElCurrentL2[1];
_s1.VoltL2 := Main_500us.VoltL2ElecDevice1;
_s1.PowFactL2 := Main_500us.PowFactL2ElecDevice1;
_s1.VoltL2_THD := Main_500us.ElectricalDevice1.stVariantValues.astLx[2].fTHD_U;
_s1.CurrentL2_THD := Main_500us.ElectricalDevice1.stVariantValues.astLx[2].fTHD_I;
_s1.CurrentL2_harm := Main_500us.ElectricalDevice1.stVariantValues.astLx[2].fHarmonics_I;
_s1.ActPowerL3 := Main_500us.ActPowL3ElecDevice1;
_s1.ReactPowerL3 := Main_500us.ReactPowL3ElecDevice1;
_s1.ApparPowerL3 := Main_500us.AppPowL3ElecDevice1;
_s1.CurrentL3 := GVL_Visu.ElCurrentL3[1];
_s1.VoltL3 := Main_500us.VoltL3ElecDevice1;
_s1.PowFactL3 := Main_500us.PowFactL3ElecDevice1;
_s1.VoltL3_THD := Main_500us.ElectricalDevice1.stVariantValues.astLx[3].fTHD_U;
_s1.CurrentL3_THD := Main_500us.ElectricalDevice1.stVariantValues.astLx[3].fTHD_I;
_s1.CurrentL3_harm := Main_500us.ElectricalDevice1.stVariantValues.astLx[3].fHarmonics_I;
SyncPulseElecDevice1(IN := GVL_Visu.MotorRunning[1], PT := T#500ms); // TP
ElectricalDevice[1](
    LineName := GVL_const.LineName,
    MachineName := GVL_const.MachineName,
    DeviceName := GVL_const.ElecDevice1,
    TimeStamp := GVL_SW.Unix_TimeStamp,
    DeviceElectricalData := _s1,
    DeviceRunning := GVL_Visu.MotorRunning[1],
    SynchPulse := SyncPulseElecDevice1.Q,
    Enable := GVL_Visu.LineRunning); // ElectricalDevicePeriodicOper
ElectPeriodicDeviceStruct01 := ElectricalDevice[1].OpcUaVal;

// PAGE Electrical Motor2 ---
// compose _s2 : ElectrDataEthCAT
_s2.ActPowerTot := Main_500us.ElectricalDevice2.stVariantValues.stTotal.fPtot;
_s2.ReactPowerTot := Main_500us.ElectricalDevice2.stVariantValues.stTotal.fQtot;
_s2.ApparPowerTot := Main_500us.ElectricalDevice2.stVariantValues.stTotal.fStot;
_s2.PowerFact := Main_500us.ElectricalDevice2.stVariantValues.stTotal.fPower_Factor;
_s2.PQF := Main_500us.ElectricalDevice2.stVariantValues.stTotal.fPQF;
_s2.ActPowerL1 := Main_500us.ActPowL1ElecDevice2;
_s2.ReactPowerL1 := Main_500us.ReactPowL1ElecDevice2;
_s2.ApparPowerL1 := Main_500us.AppPowL1ElecDevice2;
_s2.CurrentL1 := GVL_Visu.ElCurrentL1[2];
_s2.VoltL1 := Main_500us.VoltL1ElecDevice2;
_s2.PowFactL1 := Main_500us.PowFactL1ElecDevice2;
_s2.VoltL1_THD := Main_500us.ElectricalDevice2.stVariantValues.astLx[1].fTHD_U;
_s2.CurrentL1_THD := Main_500us.ElectricalDevice2.stVariantValues.astLx[1].fTHD_I;
_s2.CurrentL1_harm := Main_500us.ElectricalDevice2.stVariantValues.astLx[1].fHarmonics_I;
_s2.ActPowerL2 := Main_500us.ActPowL2ElecDevice2;
_s2.ReactPowerL2 := Main_500us.ReactPowL2ElecDevice2;
_s2.ApparPowerL2 := Main_500us.AppPowL2ElecDevice2;
_s2.CurrentL2 := GVL_Visu.ElCurrentL2[2];
_s2.VoltL2 := Main_500us.VoltL2ElecDevice2;
_s2.PowFactL2 := Main_500us.PowFactL2ElecDevice2;
_s2.VoltL2_THD := Main_500us.ElectricalDevice2.stVariantValues.astLx[2].fTHD_U;
_s2.CurrentL2_THD := Main_500us.ElectricalDevice2.stVariantValues.astLx[2].fTHD_I;
_s2.CurrentL2_harm := Main_500us.ElectricalDevice2.stVariantValues.astLx[2].fHarmonics_I;
_s2.ActPowerL3 := Main_500us.ActPowL3ElecDevice2;
_s2.ReactPowerL3 := Main_500us.ReactPowL3ElecDevice2;
_s2.ApparPowerL3 := Main_500us.AppPowL3ElecDevice2;
_s2.CurrentL3 := GVL_Visu.ElCurrentL3[2];
_s2.VoltL3 := Main_500us.VoltL3ElecDevice2;
_s2.PowFactL3 := Main_500us.PowFactL3ElecDevice2;
_s2.VoltL3_THD := Main_500us.ElectricalDevice2.stVariantValues.astLx[3].fTHD_U;
_s2.CurrentL3_THD := Main_500us.ElectricalDevice2.stVariantValues.astLx[3].fTHD_I;
_s2.CurrentL3_harm := Main_500us.ElectricalDevice2.stVariantValues.astLx[3].fHarmonics_I;
SyncPulseElecDevice2(IN := GVL_Visu.MotorRunning[2], PT := T#500ms); // TP
// Read electrical data from EL3443 module and send  it by MQTT during device RUN state.
// It allows analytics of periodically switched device
ElectricalDevice[2](
    lineName := GVL_const.LineName,
    machineName := GVL_const.MachineName,
    DeviceName := GVL_const.ElecDevice2,
    TimeStamp := GVL_SW.Unix_TimeStamp,
    DeviceElectricalData := _s2,
    DeviceRunning := GVL_Visu.MotorRunning[2],
    SynchPulse := SyncPulseElecDevice2.Q,
    Enable := GVL_Visu.LineRunning); // ElectricalDevicePeriodicOper
ElectPeriodicDeviceStruct02 := ElectricalDevice[2].OpcUaVal;
// Main_500us.rCurrL1_BC1: input not connected
// Main_500us.rCurrL2_BC1: input not connected
// Main_500us.rCurrL3_BC1: input not connected
// Main_500us.rCurrL1_BC2: input not connected
// Main_500us.rCurrL2_BC2: input not connected
// Main_500us.rCurrL3_BC2: input not connected

END_PROGRAM

// ---- POUs/FB/OPC_UA/ElectricalDevicePeriodicOper.TcPOU
FUNCTION_BLOCK ElectricalDevicePeriodicOper
VAR_INPUT
	LineName					: STRING(40);
	MachineName 				: STRING(40);
	DeviceName					: STRING(40);
	TimeStamp					: ULINT;
	DeviceElectricalData 		: ElectrDataEthCAT;
	DeviceRunning				: BOOL;
	SynchPulse					: BOOL;
	Enable						: BOOL;
END_VAR
VAR_OUTPUT
	OpcUaVal					: ElectrDevicePeriodicOper_DataModel;
END_VAR
VAR
	SetParameter 				: BOOL := TRUE;
		
	// state machine
	nState						: INT;		
	
	// structure for data exchange
	stValues					: ElectrDevicePeriodicOper_DataModel;	
	
	// Trigger for updating output OPC UA data
	UpdateOpcUa					: BOOL;
	
	// device state detection
	rtrigDeviceRunning: R_TRIG;
	ftrigDeviceRunning: F_TRIG;

	// state of monitored electrical device
	DeviceState			: BOOL;

	// safety watchdog
	tonWatchdog : TON;	
	
	StoppingCntr 	: INT;
	StoppedCntr 	: INT;
	
	 // Drive States
     RunningState	: BOOL := FALSE;
     StoppingState	: BOOL := FALSE;
     StoppedState	: BOOL := FALSE;
	 DriveStates	: DriveState_DataModel; 
END_VAR

(*
This FB evaluates electrical data from EL3443 when electrical device is in 'Running'
and creates output struct for OPC UA
*)

IF Enable THEN
		DeviceState := DeviceRunning;
		
		// synchronisation pulse from FB input
		stValues.SynchPulse := SynchPulse;
		
		// edge detection for drive state evaluation
		rtrigDeviceRunning(CLK:=DeviceState);	
		ftrigDeviceRunning(CLK:=DeviceState);	
		
		IF SetParameter THEN
			SetParameter := FALSE;		
			// constant entry in json payload
			stValues.LineName := LineName;
			stValues.MachineName := MachineName;
			stValues.DeviceName := DeviceName;
		END_IF
		
		
		// evaluate device state
		CASE nState OF
		0:
		// IDLE
			StoppingCntr 		:= 0;
			StoppedCntr 		:= 0;
			RunningState 		:= FALSE;
			StoppingState	 	:= FALSE;
			StoppedState 		:= FALSE;
			UpdateOpcUa			:= FALSE;
			stValues.DeviceState := DriveStates.StoppedState;
			
			IF rtrigDeviceRunning.Q THEN
				// sequence watchdog
				tonWatchdog.IN := TRUE; 
				nState := 10;
			END_IF
			
		10:
		// RUNNING
			RunningState := TRUE;
			stValues.DeviceState := DriveStates.RunningState;
			
			// update OPC UA values
			UpdateOpcUa := TRUE;
			
			IF ftrigDeviceRunning.Q THEN
				RunningState := FALSE;
				nState := 20;
			END_IF
		
		20:
		// STOPPING
			StoppingState 			:= TRUE;
			stValues.DeviceState 	:= DriveStates.StoppingState;
			tonWatchdog.IN := FALSE;
			
			IF StoppingState THEN StoppingCntr := StoppingCntr + 1; END_IF
			
			IF StoppingCntr = 3 THEN
				StoppingState := FALSE;
				nState := 30;
			END_IF
		
		30:
		// STOPPED
			StoppedState 			:= TRUE;
			stValues.DeviceState 	:= DriveStates.StoppedState;
		
			IF StoppedState THEN StoppedCntr := StoppedCntr + 1; END_IF
			
			IF StoppedCntr = 2 THEN
				StoppedState := FALSE;
				UpdateOpcUa := FALSE;
				nState := 0;
			END_IF
			
		END_CASE
		
		
		IF UpdateOpcUa THEN
			//write electrical data from FB input to OPC UA structure
			stValues.ElectricalData := DeviceElectricalData;
			stValues.TimeStamp := TimeStamp;
			OpcUaVal := stValues;
		END_IF
ELSE
		tonWatchdog.IN := FALSE;
		nState := 0;
END_IF

IF tonWatchdog.ET > T#10S THEN
	nState := 0;
END_IF
tonWatchdog(PT:=T#10S);

END_FUNCTION_BLOCK

// ---- POUs/PRG_500us/Main_500us.TcPOU
PROGRAM Main_500us
VAR
	ElectricalDevice1 					: FB_EL3443;		// electrical device e.g. motor, drive
	ElectricalDevice2 					: FB_EL3443;		// electrical device e.g. motor, drive
	
	// electrical device 1, phase L1
	CurrL1ElecDevice1					: REAL;
	VoltL1ElecDevice1					: REAL;
	ActPowL1ElecDevice1					: REAL;
	AppPowL1ElecDevice1					: REAL;
	ReactPowL1ElecDevice1				: REAL;
	PowFactL1ElecDevice1				: REAL;
	
	// electrical device 1, phase L2
	CurrL2ElecDevice1					: REAL;
	VoltL2ElecDevice1					: REAL;
	ActPowL2ElecDevice1					: REAL;
	AppPowL2ElecDevice1					: REAL;
	ReactPowL2ElecDevice1				: REAL;
	PowFactL2ElecDevice1				: REAL;
	
	// electrical device 1, phase L3
	CurrL3ElecDevice1					: REAL;
	VoltL3ElecDevice1					: REAL;
	ActPowL3ElecDevice1					: REAL;
	AppPowL3ElecDevice1					: REAL;
	ReactPowL3ElecDevice1				: REAL;
	PowFactL3ElecDevice1				: REAL;

	// electrical device 2, phase L1
	CurrL1ElecDevice2					: REAL;
	VoltL1ElecDevice2					: REAL;
	ActPowL1ElecDevice2					: REAL;
	AppPowL1ElecDevice2					: REAL;
	ReactPowL1ElecDevice2				: REAL;
	PowFactL1ElecDevice2				: REAL;
	
	// electrical device 2, phase L2
	CurrL2ElecDevice2					: REAL;
	VoltL2ElecDevice2					: REAL;
	ActPowL2ElecDevice2					: REAL;
	AppPowL2ElecDevice2					: REAL;
	ReactPowL2ElecDevice2				: REAL;
	PowFactL2ElecDevice2				: REAL;
	
	// electrical device 2, phase L3
	CurrL3ElecDevice2					: REAL;
	VoltL3ElecDevice2					: REAL;
	ActPowL3ElecDevice2					: REAL;
	AppPowL3ElecDevice2					: REAL;
	ReactPowL3ElecDevice2				: REAL;
	PowFactL3ElecDevice2				: REAL;
	
		
END_VAR

(* 
This PRG should run in very fast task (500us) to enable 
proper real-time data acquisition from EL3443 measurement modules.
*)

ElectricalDevice1(
	bEnable:= TRUE , 
	stStatusTotal=> , 
	stStatusPhase_L1=> , 
	stStatusPhase_L2=> , 
	stStatusPhase_L3=> , 
	stVariantValues=> , 
	bError=> );
	
ElectricalDevice2(
	bEnable:= TRUE , 
	stStatusTotal=> , 
	stStatusPhase_L1=> , 
	stStatusPhase_L2=> , 
	stStatusPhase_L3=> , 
	stVariantValues=> , 
	bError=> );
	

	
	// data from IO proces image - very fast (real time)
	CurrL1ElecDevice1 	:= ElectricalDevice1.stEL3443_IO.MDP5001_341_Input.MDP5001_341_L1_Basic_Current;
	VoltL1ElecDevice1 	:= ElectricalDevice1.stEL3443_IO.MDP5001_341_Input.MDP5001_341_L1_Basic_Voltage;
	ActPowL1ElecDevice1 	:= ElectricalDevice1.stEL3443_IO.MDP5001_341_Input.MDP5001_341_L1_Power_Active_Power;
	AppPowL1ElecDevice1 	:= ElectricalDevice1.stEL3443_IO.MDP5001_341_Input.MDP5001_341_L1_Power_Apparent_Power;
	ReactPowL1ElecDevice1 := ElectricalDevice1.stEL3443_IO.MDP5001_341_Input.MDP5001_341_L1_Power_Reactive_Power;
	PowFactL1ElecDevice1 	:= ElectricalDevice1.stEL3443_IO.MDP5001_341_Input.MDP5001_341_L1_Power_Power_Factor;
	
	CurrL2ElecDevice1 	:= ElectricalDevice1.stEL3443_IO.MDP5001_341_Input.MDP5001_341_L2_Basic_Current;
	VoltL2ElecDevice1 	:= ElectricalDevice1.stEL3443_IO.MDP5001_341_Input.MDP5001_341_L2_Basic_Voltage;
	ActPowL2ElecDevice1 	:= ElectricalDevice1.stEL3443_IO.MDP5001_341_Input.MDP5001_341_L2_Power_Active_Power;
	AppPowL2ElecDevice1 	:= ElectricalDevice1.stEL3443_IO.MDP5001_341_Input.MDP5001_341_L2_Power_Apparent_Power;
	ReactPowL2ElecDevice1 := ElectricalDevice1.stEL3443_IO.MDP5001_341_Input.MDP5001_341_L2_Power_Reactive_Power;
	PowFactL2ElecDevice1 	:= ElectricalDevice1.stEL3443_IO.MDP5001_341_Input.MDP5001_341_L2_Power_Power_Factor;
	
	CurrL3ElecDevice1 	:= ElectricalDevice1.stEL3443_IO.MDP5001_341_Input.MDP5001_341_L3_Basic_Current;
	VoltL3ElecDevice1 	:= ElectricalDevice1.stEL3443_IO.MDP5001_341_Input.MDP5001_341_L3_Basic_Voltage;
	ActPowL3ElecDevice1 	:= ElectricalDevice1.stEL3443_IO.MDP5001_341_Input.MDP5001_341_L3_Power_Active_Power;
	AppPowL3ElecDevice1 	:= ElectricalDevice1.stEL3443_IO.MDP5001_341_Input.MDP5001_341_L3_Power_Apparent_Power;
	ReactPowL3ElecDevice1 := ElectricalDevice1.stEL3443_IO.MDP5001_341_Input.MDP5001_341_L3_Power_Reactive_Power;
	PowFactL3ElecDevice1 	:= ElectricalDevice1.stEL3443_IO.MDP5001_341_Input.MDP5001_341_L3_Power_Power_Factor;
	
	CurrL1ElecDevice2 	:= ElectricalDevice2.stEL3443_IO.MDP5001_341_Input.MDP5001_341_L1_Basic_Current;
	VoltL1ElecDevice2 	:= ElectricalDevice2.stEL3443_IO.MDP5001_341_Input.MDP5001_341_L1_Basic_Voltage;
	ActPowL1ElecDevice2 	:= ElectricalDevice2.stEL3443_IO.MDP5001_341_Input.MDP5001_341_L1_Power_Active_Power;
	AppPowL1ElecDevice2 	:= ElectricalDevice2.stEL3443_IO.MDP5001_341_Input.MDP5001_341_L1_Power_Apparent_Power;
	ReactPowL1ElecDevice2 := ElectricalDevice2.stEL3443_IO.MDP5001_341_Input.MDP5001_341_L1_Power_Reactive_Power;
	PowFactL1ElecDevice2 	:= ElectricalDevice2.stEL3443_IO.MDP5001_341_Input.MDP5001_341_L1_Power_Power_Factor;
	
	CurrL2ElecDevice2 	:= ElectricalDevice2.stEL3443_IO.MDP5001_341_Input.MDP5001_341_L2_Basic_Current;
	VoltL2ElecDevice2 	:= ElectricalDevice2.stEL3443_IO.MDP5001_341_Input.MDP5001_341_L2_Basic_Voltage;
	ActPowL2ElecDevice2 	:= ElectricalDevice2.stEL3443_IO.MDP5001_341_Input.MDP5001_341_L2_Power_Active_Power;
	AppPowL2ElecDevice2 	:= ElectricalDevice2.stEL3443_IO.MDP5001_341_Input.MDP5001_341_L2_Power_Apparent_Power;
	ReactPowL2ElecDevice2 := ElectricalDevice2.stEL3443_IO.MDP5001_341_Input.MDP5001_341_L2_Power_Reactive_Power;
	PowFactL2ElecDevice2 	:= ElectricalDevice2.stEL3443_IO.MDP5001_341_Input.MDP5001_341_L2_Power_Power_Factor;
	
	CurrL3ElecDevice2 	:= ElectricalDevice2.stEL3443_IO.MDP5001_341_Input.MDP5001_341_L3_Basic_Current;
	VoltL3ElecDevice2 	:= ElectricalDevice2.stEL3443_IO.MDP5001_341_Input.MDP5001_341_L3_Basic_Voltage;
	ActPowL3ElecDevice2 	:= ElectricalDevice2.stEL3443_IO.MDP5001_341_Input.MDP5001_341_L3_Power_Active_Power;
	AppPowL3ElecDevice2 	:= ElectricalDevice2.stEL3443_IO.MDP5001_341_Input.MDP5001_341_L3_Power_Apparent_Power;
	ReactPowL3ElecDevice2 := ElectricalDevice2.stEL3443_IO.MDP5001_341_Input.MDP5001_341_L3_Power_Reactive_Power;
	PowFactL3ElecDevice2 	:= ElectricalDevice2.stEL3443_IO.MDP5001_341_Input.MDP5001_341_L3_Power_Power_Factor;
	

	
	// data from FB processing (with some delay - not really real-time)
	(*ElectricalDevice2.stVariantValues.astLx[1].fI_RMS;
	ElectricalDevice2.stVariantValues.astLx[1].fPower_Factor;
	ElectricalDevice2.stVariantValues.astLx[1].fP;
	ElectricalDevice2.stVariantValues.astLx[1].fQ;
	ElectricalDevice2.stVariantValues.astLx[1].fS;
	
	ElectricalDevice2.stVariantValues.astLx[1].fHarmonics_I;
	*)

END_PROGRAM

// ---- POUs/PRG_10ms/PRG_06_ElectricalMonitoring.TcPOU
PROGRAM PRG_06_ElectricalMonitoring
VAR
	ElectDeviceContOper					: ElectricalDeviceContOper;
	
	ElectrDeviceContOper				: ReadMBSentron_PAC1200;
	
	{attribute 'OPC.UA.DA' := '1'}
	{attribute 'OPC.UA.DA.Access' := '1'}			// read only
	{attribute 'OPC.UA.DA.StructuredType' := '1'}
	ElectContinousDeviceStruct01		: ElectrDeviceContOper_DataModel;
END_VAR

// Read electrical data over Modbus TCP from Sentron 7KT PAC1200 and send it continously by MQTT.
// IP address of Sentron device
ElectrDeviceContOper(IpAddress := '192.168.1.177', RequestTime := T#100MS, Enable := GVL_Visu.LineRunning); // ReadMBSentron_PAC1200
ElectDeviceContOper(
    LineName := GVL_const.LineName,
    MachineName := GVL_const.MachineName,
    DeviceName := GVL_const.ElecDevice3,
    TimeStamp := GVL_SW.Unix_TimeStamp,
    DeviceElectricalData := ElectrDeviceContOper.ElectricalData,
    Enable := GVL_Visu.LineRunning); // ElectricalDeviceContOper
ElectContinousDeviceStruct01 := ElectDeviceContOper.OpcUaVal;

END_PROGRAM

// ---- POUs/FB/OPC_UA/ElectricalDeviceContOper.TcPOU
FUNCTION_BLOCK ElectricalDeviceContOper
VAR_INPUT
	LineName					: STRING(40);
	MachineName 				: STRING(40);
	DeviceName					: STRING(40);
	TimeStamp					: ULINT;
	DeviceElectricalData 		: ElectrDataModbusTCP;
	Enable						: BOOL;
END_VAR
VAR_OUTPUT
	OpcUaVal					: ElectrDeviceContOper_DataModel;	
END_VAR
VAR
	SetParameter 				: BOOL := TRUE;		
	
	stValues					: ElectrDeviceContOper_DataModel;		
END_VAR

(*
This FB evaluates continously  electrical data from Sentron 7KT PAC1200 
and creates output struct for OPC UA
*)

IF Enable THEN	
		
		IF SetParameter THEN
			SetParameter := FALSE;
	
			// constant entry in json payload
			stValues.LineName := LineName;
			stValues.MachineName := MachineName;
			stValues.DeviceName := DeviceName;
		END_IF
		
		stValues.TimeStamp := TimeStamp;
		stValues.ElectricalData := DeviceElectricalData;
		OpcUaVal := stValues;
ELSE
		;
END_IF

END_FUNCTION_BLOCK

// ---- POUs/FB/ModbusTCP/ReadMBSentron_PAC1200.TcPOU
FUNCTION_BLOCK ReadMBSentron_PAC1200
VAR_INPUT
	IpAddress						: STRING(20);
	RequestTime						: TIME := T#100MS;
	Enable						: BOOL;
END_VAR
VAR CONSTANT
	wMBAddress_Read				: WORD 					:= 16#0001;								// First address to read
	wMBAddress_Write			: WORD 					:= 16#3010;								// First address to write
END_VAR
VAR	
	arReadRegs					: ARRAY [0..16#49] OF WORD;										// read 73dec WORDs via Modbus
	
	arReadRegsCycle0			: ARRAY [0..16#49] OF WORD;										// register 0..73
	arReadRegsCycle1			: ARRAY [0..16#49] OF WORD;										// register 74..145

	ErrorID						: UDINT;														// Last error
	wCounterSuccess				: WORD;
	wCounterErrors				: WORD;	
	
	// Application variables
	Step						: INT;
	tonRecycle					: TON;
	Auto						: BOOL := TRUE;													// Continuous RW
	// FBs
	fbMBReadRegs				: FB_MBReadRegs;
	fbMBWriteRegs				: FB_MBWriteRegs;
	MBcycle						: BYTE;															// cycle 0 = read registers 0..73, cycle 1 = read registers 74..145
	
	wMBAddressRead				: WORD ;														// First address to read

END_VAR
VAR_OUTPUT
	ElectricalData				: ElectrDataModbusTCP;
END_VAR

// This PRG reads 146 registers (16bit) via MODBUS function 3. 
// Due to the limitation of reading only 128 registers with FB_MBReadRegs from Beckhoff library TF6250
// there is a switching mechanism for reading registers in two cycles
// during cycle0  - registers from 0..73 are read
// during cycle1  - registers from 74..145 are read

// Timer for auto mode - Read/write frequency
tonRecycle(IN:= Auto AND NOT tonRecycle.Q, PT:= RequestTime);


CASE Step OF

	0:	// Idle

		ErrorID				:= 0;
		IF tonRecycle.Q THEN
			Step 				:= Step + 10;
		END_IF

	10:	// Read Registers - Modbus function 3

		fbMBReadRegs.bExecute 	:= TRUE;
		Step 					:= Step + 10;
		
		//set MB address for different request step
		IF MBcycle = 0 THEN
			wMBAddressRead := 16#0000;					// start reading from adress 0
		
		ELSIF MBcycle = 1 THEN
			wMBAddressRead := 16#004A;					// start reading from adress 74
		END_IF
	

	20:	// Wait till register read ends

		fbMBReadRegs.bExecute 	:= FALSE;
		IF NOT fbMBReadRegs.bBusy THEN
			IF NOT fbMBReadRegs.bError THEN
				Step 			:= Step + 10;
				
				//save data from MB to proper array
				IF MBcycle = 0 THEN
					arReadRegsCycle0 := arReadRegs;
				ELSIF MBcycle = 1 THEN
					arReadRegsCycle1 := arReadRegs;
				END_IF
				
				//increase MB step after each successful reading of MB data
				MBcycle := MBcycle+1;
				
				IF  MBcycle >1 THEN
					MBcycle :=0;
				END_IF
				
			ELSE
				ErrorID			:= fbMBReadRegs.nErrId;
				wCounterErrors	:= wCounterErrors + 1;
				Step 			:= 100;
			END_IF
		END_IF

	30:	// Write Registers - Modbus function 16

		//fbMBWriteRegs.bExecute 	:= TRUE;
		//iStep 					:= iStep + 10;
		
		Step := 0;	//only test, delete it
		
	40:	
		

		// Wait till register write ends
		(*
		fbMBWriteRegs.bExecute 	:= FALSE;
		IF NOT fbMBWriteRegs.bBusy THEN
			IF NOT fbMBWriteRegs.bError THEN
				wCounterSuccess	:= wCounterSuccess + 1;
				iStep 			:= 0;
			ELSE
				udiErrorID		:= fbMBWriteRegs.nErrId;
				wCounterErrors	:= wCounterErrors + 1;
				iStep 			:= 100;
			END_IF
		END_IF
		*)

	100: // Error
		Step := 0;
		;

END_CASE

// Read Modbus function 3
fbMBReadRegs(	sIPAddr			:= IpAddress, 
				nTCPPort		:= MODBUS_TCP_PORT,
				nQuantity		:= SIZEOF(arReadRegs)/2,								//SIZEOF(arrReadRegs)/2, 
				nMBAddr			:= wMBAddressRead, 
				cbLength		:= SIZEOF(arReadRegs),									//SIZEOF(arrReadRegs), 
				pDestAddr		:= ADR(arReadRegs));
				

// output electrical data
ElectricalData.ActPowerPos := DWORD_TO_REAL((arReadRegsCycle0[0] * 65536) + arReadRegsCycle0[1] ) * 0.1/1000.0;			// Total + Active power [kW]
ElectricalData.ActPowerNeg := DWORD_TO_REAL((arReadRegsCycle0[2] * 65536) + arReadRegsCycle0[3] ) * 0.1/1000.0;			// Total - Active power [kW]

ElectricalData.ReactPowerPos := DWORD_TO_REAL((arReadRegsCycle0[4] * 65536) + arReadRegsCycle0[5]) * 0.1/1000.0;		// Total + Reactive power [kvar]
ElectricalData.ReactPowerNeg := DWORD_TO_REAL((arReadRegsCycle0[6] * 65536) + arReadRegsCycle0[7]) * 0.1/1000.0;		// Total - Reactive power [kvar]

ElectricalData.ApparPowerPos := DWORD_TO_REAL((arReadRegsCycle0[16] * 65536) + arReadRegsCycle0[17]) * 0.1/1000.0;		// Total + Apparent power [kVA]
ElectricalData.ApparPowerNeg := DWORD_TO_REAL((arReadRegsCycle0[18] * 65536) + arReadRegsCycle0[19]) * 0.1/1000.0;		// Total - Apparent power [kVA]

ElectricalData.PowerFact 	:= WORD_TO_REAL(arReadRegsCycle0[25]) * 0.001 ;		// Power factor total [no unit]
ElectricalData.LineFreq		:= WORD_TO_REAL(arReadRegsCycle0[27]) * 0.001 ;		// Line frequency [Hz]


// L1 electrical data
ElectricalData.ActPowerPosL1 := DWORD_TO_REAL((arReadRegsCycle0[40] * 65536) + arReadRegsCycle0[41]) * 0.1/1000.0;		// + Active power L1 [kW]
ElectricalData.ActPowerNegL1 := DWORD_TO_REAL((arReadRegsCycle0[42] * 65536) + arReadRegsCycle0[43]) * 0.1/1000.0;		// - Active power L1 [kW]

ElectricalData.ReactPowerPosL1 := DWORD_TO_REAL((arReadRegsCycle0[44] * 65536) + arReadRegsCycle0[45]) * 0.1/1000.0;	// + Reactive power L1 [kW]
ElectricalData.ReactPowerNegL1 := DWORD_TO_REAL((arReadRegsCycle0[46] * 65536) + arReadRegsCycle0[47]) * 0.1/1000.0;	// - Reactive power L1 [kW]

ElectricalData.CurrentL1 := DWORD_TO_REAL((arReadRegsCycle0[60] * 65536) + arReadRegsCycle0[61]) * 0.001;				// Current L1 [A]
ElectricalData.PowFactL1 := WORD_TO_REAL(arReadRegsCycle0[65]) * 0.001 ;												// Power factor L1 [no unit]

// L2 electrical data
ElectricalData.ActPowerPosL2 := DWORD_TO_REAL((arReadRegsCycle1[6] * 65536) + arReadRegsCycle1[7]) * 0.1/1000.0;		// + Active power L2 [kW]
ElectricalData.ActPowerNegL2 := DWORD_TO_REAL((arReadRegsCycle1[8] * 65536) + arReadRegsCycle1[9]) * 0.1/1000.0;		// - Active power L2 [kW]

ElectricalData.ReactPowerPosL2 := DWORD_TO_REAL((arReadRegsCycle1[10] * 65536) + arReadRegsCycle1[11]) * 0.1/1000.0;	// + Reactive power L2 [kW] 
ElectricalData.ReactPowerNegL2 := DWORD_TO_REAL((arReadRegsCycle1[12] * 65536) + arReadRegsCycle1[13]) * 0.1/1000.0;	// - Reactive power L2 [kW]

ElectricalData.CurrentL2 := DWORD_TO_REAL((arReadRegsCycle1[26] * 65536) + arReadRegsCycle1[27]) * 0.001;				// Current L2 [A]
ElectricalData.PowFactL2 := WORD_TO_REAL(arReadRegsCycle0[31]) * 0.001;													// Power factor L2 [no unit]										

// L3 electrical data
ElectricalData.ActPowerPosL3 := DWORD_TO_REAL((arReadRegsCycle1[46] * 65536) + arReadRegsCycle1[47]) * 0.1/1000.0;		// + Active power L3 [kW]
ElectricalData.ActPowerNegL3 := DWORD_TO_REAL((arReadRegsCycle1[48] * 65536) + arReadRegsCycle1[49]) * 0.1/1000.0;		// - Active power L3 [kW]
 
ElectricalData.ReactPowerPosL3 := DWORD_TO_REAL((arReadRegsCycle1[50] * 65536) + arReadRegsCycle1[51]) * 0.1/1000.0;	// + Reactive power L3 [kW]
ElectricalData.ReactPowerNegL3 := DWORD_TO_REAL((arReadRegsCycle1[52] * 65536) + arReadRegsCycle1[53]) * 0.1/1000.0;	// - Reactive power L3 [kW]
 
ElectricalData.CurrentL3 := DWORD_TO_REAL((arReadRegsCycle1[66] * 65536) + arReadRegsCycle1[67]) * 0.001;				// Current L3 [A]
ElectricalData.PowFactL3 := WORD_TO_REAL(arReadRegsCycle0[71]) * 0.001 ;												// Power factor L3 [no unit]

END_FUNCTION_BLOCK

// ---- POUs/PRG_10ms/PRG_07_LineState.TcPOU
PROGRAM PRG_07_LineState
VAR
	CheckLine1Producing	: CheckLineProducing;
	
	ValueChangeDetector	:	ARRAY[1..6] OF ValueChangeDetector;
	GenericState		:	ARRAY[1..6] OF GenericState;
	tpValueChangeDelay	:	ARRAY[1..6] OF TP;
	
	{attribute 'OPC.UA.DA' := '1'}
	{attribute 'OPC.UA.DA.Access' := '1'}			// read only
	{attribute 'OPC.UA.DA.StructuredType' := '1'}
	AutoModeStruct						: SingleState_DataModel;
	
	{attribute 'OPC.UA.DA' := '0'}
	{attribute 'OPC.UA.DA.Access' := '1'}			// read only
	{attribute 'OPC.UA.DA.StructuredType' := '1'}
	DoorOpenedStruct					: SingleState_DataModel;
	
	{attribute 'OPC.UA.DA' := '0'}
	{attribute 'OPC.UA.DA.Access' := '1'}			// read only
	{attribute 'OPC.UA.DA.StructuredType' := '1'}
	LineProducingStruct					: SingleState_DataModel;
	
END_VAR


// PAGE Check if line is producing --
CheckLine1Producing(OkProductNumber := GVL_Visu.OkProductCount); // CheckLineProducing
GVL_Visu.LineProducing := CheckLine1Producing.LineProducing;

// PAGE Send line states over MQTT ---
ValueChangeDetector[1](Value := BOOL_TO_INT(GVL_Visu.AutoMode)); // ValueChangeDetector
tpValueChangeDelay[1](IN := ValueChangeDetector[1].ValueChanged, PT := T#50MS); // TP
GenericState[1](
    LineName := GVL_const.LineName,
    MachineName := GVL_const.MachineName,
    StateName := 'AutoMode',
    TimeStamp := GVL_SW.Unix_TimeStamp,
    Value := BOOL_TO_INT(GVL_Visu.AutoMode),
    Enable := tpValueChangeDelay[1].Q); // GenericState
AutoModeStruct := GenericState[1].OpcUaVal;
ValueChangeDetector[2](Value := BOOL_TO_INT(GVL_Visu.AutoMode)); // ValueChangeDetector
tpValueChangeDelay[2](IN := ValueChangeDetector[2].ValueChanged, PT := T#50MS); // TP
GenericState[2](
    LineName := GVL_const.LineName,
    MachineName := GVL_const.MachineName,
    StateName := 'DoorOpened',
    TimeStamp := GVL_SW.Unix_TimeStamp,
    Value := BOOL_TO_INT(GVL_Visu.AutoMode),
    Enable := tpValueChangeDelay[2].Q); // GenericState
DoorOpenedStruct := GenericState[2].OpcUaVal;
ValueChangeDetector[3](Value := BOOL_TO_INT(GVL_Visu.LineProducing)); // ValueChangeDetector
tpValueChangeDelay[3](IN := ValueChangeDetector[3].ValueChanged, PT := T#50MS); // TP
GenericState[3](
    LineName := GVL_const.LineName,
    MachineName := GVL_const.MachineName,
    StateName := 'LineProducing',
    TimeStamp := GVL_SW.Unix_TimeStamp,
    Value := BOOL_TO_INT(GVL_Visu.LineProducing),
    Enable := tpValueChangeDelay[3].Q); // GenericState
LineProducingStruct := GenericState[3].OpcUaVal;
ValueChangeDetector[4](Value := UINT_TO_INT(GVL_Visu.OkProductCount)); // ValueChangeDetector

END_PROGRAM

// ---- POUs/FB/Generic/CheckLineProducing.TcPOU
FUNCTION_BLOCK CheckLineProducing
VAR_INPUT
	OkProductNumber		: UINT;
	NokProductNumber	: UINT;
END_VAR
VAR_OUTPUT
	LineProducing		: BOOL;
END_VAR
VAR
	ProductOK			: UINT;
	ProductNok			: UINT;
	ProductOkMem		: UINT;
	ProductNokMem		: UINT;
	
	LineStoppedMem		: BOOL;
	tonLineStopped		: TON;
	LineStopped			: SR;
	LineInOperation		: SR;
END_VAR

(*
This FB checks if line is producing by evaluation of product pieces. 
If product pieces number is increasing within time window
it means line is producing.
*) 

ProductOK :=OkProductNumber;
ProductNok := NokProductNumber;

LineStoppedMem := ProductOK=ProductOkMem;

tonLineStopped(IN:=LineStoppedMem , PT:=T#10S , Q=> , ET=> );

IF ProductOK <> ProductOkMem THEN
	ProductOkMem := ProductOK; 
END_IF

LineStopped(SET1:=tonLineStopped.Q , RESET:=NOT tonLineStopped.Q , Q1=> );
LineInOperation(SET1:= NOT tonLineStopped.Q, RESET:=tonLineStopped.Q , Q1=> );

LineProducing := LineInOperation.Q1;

END_FUNCTION_BLOCK

// ---- POUs/FB/Generic/ValueChangeDetector.TcPOU
FUNCTION_BLOCK ValueChangeDetector
VAR_INPUT
	Value			:	INT;
END_VAR
VAR_OUTPUT
	ValueChanged	:	BOOL;
END_VAR
VAR
	ValueCurrent	:	INT;
	ValueMem		:	INT;
	SetInit			:	BOOL := TRUE;
END_VAR

(*
Detect value change
*)

ValueCurrent := Value;

ValueChanged := ValueCurrent<>ValueMem;

ValueMem:=ValueCurrent;

// set once to changed on init cycle
// it allows to send data after power recycle 
IF SetInit THEN
	SetInit := FALSE;
	ValueChanged := TRUE;
END_IF

END_FUNCTION_BLOCK

// ---- POUs/FB/OPC_UA/GenericState.TcPOU
FUNCTION_BLOCK GenericState
VAR_INPUT
	LineName	: STRING(40);
	MachineName : STRING(40);
	StateName	: STRING(40);
	TimeStamp	: ULINT;
	Value		: INT;	 
	Enable		: BOOL; 		//enable state evaluation
END_VAR
VAR_OUTPUT
	OpcUaVal		: SingleState_DataModel;
END_VAR
VAR
	SetParameter : BOOL := TRUE;	
	
	stValues		: SingleState_DataModel;	
	
	// safety watchdog
	tonWatchdog : TON;
END_VAR

(*
This FB evaluates any state value and creates output struct for OPC UA
*) 

IF Enable THEN
	
	IF SetParameter THEN
		SetParameter := FALSE;
		// constant entry
		stValues.LineName := LineName;
		stValues.MachineName := MachineName;
		stValues.StateName := StateName;
	END_IF
	
	stValues.TimeStamp := TimeStamp;
	stValues.StateValue := Value;
		
	OpcUaVal := stValues;
ELSE
	;
END_IF;

END_FUNCTION_BLOCK

// ---- POUs/PRG_10ms/PRG_08_ProductionStatistics.TcPOU
PROGRAM PRG_08_ProductionStatistics
VAR
	PartsPerMinInstant					: PartsPerMinInstant2;
	PartsPerMin							: GenericState;
	OkPartsPerMinHistorical				: PartsPerMinHistorical;
	
	{attribute 'OPC.UA.DA' := '1'}
	{attribute 'OPC.UA.DA.Access' := '1'}			// read only
	{attribute 'OPC.UA.DA.StructuredType' := '1'}
	OkPartsPerMinStruct					: SingleState_DataModel;
END_VAR

PartsPerMinInstant(TotalCount := GVL_Visu.OkProductCount); // PartsPerMinInstant2
GVL_Visu.OkPartsPerMinRate := PartsPerMinInstant.PPM;
PartsPerMin(
    LineName := GVL_const.LineName,
    MachineName := GVL_const.MachineName,
    StateName := 'PartsPerMinute',
    TimeStamp := GVL_SW.Unix_TimeStamp,
    Value := TO_INT(PartsPerMinInstant.PPM),
    Enable := GVL_Visu.LineRunning); // GenericState
OkPartsPerMinStruct := PartsPerMin.OpcUaVal;
OkPartsPerMinHistorical(ProductSensor := GVL_Visu.SensorProductActive, PartsPerMinHist := GVL_Visu.OkPartsPerMinHistorical); // PartsPerMinHistorical

END_PROGRAM

// ---- POUs/FB/Generic/PartsPerMinInstant.TcPOU
FUNCTION_BLOCK PartsPerMinInstant
VAR_INPUT
	// product total count
	TotalCount					: UINT;
	//Time in sec. to monitor of TotalCount changes 
	MonitorTimeSec				: UINT := 10;
END_VAR
VAR_OUTPUT
	// Parts per minut ratio
	PPM							: UINT;
END_VAR
VAR
	InitBit						:	BOOL:=TRUE;

	CurrentTotalCount			: 	UINT;
	OldTotalCount				:	UINT;
	tonRecycle					:	TON;
	rtrigCycleElapsed			:	R_TRIG;
	CountDiff					:	UINT;
END_VAR

(*
This FB calculates instantaneous parts per minute rate.
It counts TotalCount changes within 'MonitorTimeSec' window (default 10sec).
TotalCount 		-	 total number of counted products 
MonitorTimeSec	-	 monitoring time in seconds
*)

IF InitBit THEN
	CurrentTotalCount:=TotalCount;
	InitBit:=FALSE;
END_IF

tonRecycle(IN:=NOT tonRecycle.Q, PT:=UINT_TO_TIME(MonitorTimeSec * 1000));
rtrigCycleElapsed(CLK:=tonRecycle.Q);

CurrentTotalCount := TotalCount;

IF rtrigCycleElapsed.Q THEN
	CountDiff := CurrentTotalCount - OldTotalCount;
	OldTotalCount := CurrentTotalCount;
END_IF

// recalculate to 60 sec. (1min)
PPM :=  TO_UINT((60.0 / TO_REAL(MonitorTimeSec)) * TO_REAL(CountDiff));

END_FUNCTION_BLOCK

// ---- POUs/FB/Generic/PartsPerMinInstant2.TcPOU
FUNCTION_BLOCK PartsPerMinInstant2
VAR_INPUT
	// product total count
	TotalCount		: UINT;
END_VAR
VAR_OUTPUT
	// Parts per minut ratio
	PPM							: UINT;
END_VAR
VAR
	InitBit						: BOOL;
	OldTotalCount				: UINT;
	CountDiff					: UINT;
	rtrigTotalCountChanged		: R_TRIG;
	TotalCountChanged			: BOOL;
	SeqState					: INT := 0;
	tonPulseTimer				: TON;
	PulseTime					: TIME;
END_VAR

(*
This FB calculates instantaneous parts per minute rate.
It counts pulse time between TotalCount changes. 
TotalCount 		-	 total number of counted products 
*)
IF InitBit THEN
	OldTotalCount := TotalCount;
	InitBit:=FALSE;
END_IF

TotalCountChanged := FALSE;

IF TotalCount > OldTotalCount THEN
	TotalCountChanged := TRUE;
	CountDiff := TotalCount - OldTotalCount;
END_IF;
OldTotalCount := TotalCount;

rtrigTotalCountChanged(CLK:=TotalCountChanged);

CASE SeqState OF
	0:
		IF rtrigTotalCountChanged.Q THEN
			tonPulseTimer.IN:=TRUE;
			SeqState := 10;
		END_IF
	10:
		IF rtrigTotalCountChanged.Q THEN
			PulseTime := tonPulseTimer.ET;
			tonPulseTimer.IN:=FALSE;
			SeqState := 20;
		END_IF
	20:
		tonPulseTimer.IN:=TRUE;
		SeqState := 10;
END_CASE;

tonPulseTimer(PT:=T#10M);

IF TO_INT(PulseTime) <> 0 THEN
	PPM := TO_UINT(TO_REAL(60 * CountDiff) / (TIME_TO_REAL(PulseTime)/1000.0));
END_IF;

END_FUNCTION_BLOCK

// ---- POUs/FB/Generic/PartsPerMinHistorical.TcPOU
FUNCTION_BLOCK PartsPerMinHistorical
VAR_INPUT
	// Sensor activated when product counted
	ProductSensor		:	BOOL;
END_VAR
VAR_IN_OUT
	PartsPerMinHist		:	ARRAY[1..5] OF INT;
END_VAR
VAR
	tonTimer			:	TON;
	rtTimeElapsed		:	R_TRIG;
	rtProductCounted	:	R_TRIG;
	ProductCount		:	INT;
	Idx					:	INT;
END_VAR

(*
This FB calculates number of counted products within one minute.
It includes historical data.
After one minute elapses, current value from index 5 of array 
is moved to next index on the left.  Other indexes are also moved to the left.
This way the array can be used for HMI chart showing data production from 
last 5 minutes  
*)
tonTimer(IN:= NOT tonTimer.Q, PT:= T#60S);

rtProductCounted(CLK:=ProductSensor);
IF rtProductCounted.Q THEN ProductCount := ProductCount+1; END_IF;

PartsPerMinHist[5] := ProductCount;

rtTimeElapsed(CLK:=tonTimer.Q);
IF rtTimeElapsed.Q THEN
	FOR Idx := 1 TO 4 BY 1 DO
		PartsPerMinHist[Idx]:=PartsPerMinHist[Idx+1];
	END_FOR
	ProductCount := 0;
END_IF

END_FUNCTION_BLOCK

// ---- POUs/PRG_10ms/PRG_09_PlcDiagnostic.TcPOU
PROGRAM PRG_09_PlcDiagnostic
VAR
	NetID						: 	STRING := '192.168.1.145.1.1';
	tonRecycle50ms				: 	TON;
	tonRecyclePublishMqtt		: 	TON;
	
	CpuMemoryUsage				:	ReadMemoryUsage;
	CpuUsageEx_Core2			:	TC_CPuUsageEx;
	CpuUsageEx_Core3			:	TC_CPuUsageEx;
	CpuLatencyEx_Core2			:	TC_SysLatencyEx;
	CpuLatencyEx_Core3			:	TC_SysLatencyEx;
	
	PlcDiagState				:	ARRAY [1..5] OF GenericState;
	
	{attribute 'OPC.UA.DA' := '0'}
	{attribute 'OPC.UA.DA.Access' := '1'}			// read only
	{attribute 'OPC.UA.DA.StructuredType' := '1'}
	PlcCpuMemUsageStruct		: SingleState_DataModel;
	
	{attribute 'OPC.UA.DA' := '0'}
	{attribute 'OPC.UA.DA.Access' := '1'}			// read only
	{attribute 'OPC.UA.DA.StructuredType' := '1'}
	PlcCpuCore2UsageStruct		: SingleState_DataModel;
	
	{attribute 'OPC.UA.DA' := '0'}
	{attribute 'OPC.UA.DA.Access' := '1'}			// read only
	{attribute 'OPC.UA.DA.StructuredType' := '1'}
	PlcCpuCore3UsageStruct		: SingleState_DataModel;
	
	{attribute 'OPC.UA.DA' := '0'}
	{attribute 'OPC.UA.DA.Access' := '1'}			// read only
	{attribute 'OPC.UA.DA.StructuredType' := '1'}
	PlcCpuCore2JitterStruct		: SingleState_DataModel;
	
	{attribute 'OPC.UA.DA' := '0'}
	{attribute 'OPC.UA.DA.Access' := '1'}			// read only
	{attribute 'OPC.UA.DA.StructuredType' := '1'}
	PlcCpuCore3JitterStruct		: SingleState_DataModel;

END_VAR


// PAGE Recycle Timers for general usage ---
tonRecyclePublishMqtt(IN := NOT tonRecyclePublishMqtt.Q, PT := T#2s); // TON
tonRecycle50ms(IN := NOT tonRecycle50ms.Q, PT := T#50ms); // TON

// PAGE PLC Memory usage ---
PlcCpuMemUsageStruct := PlcDiagState[1].OpcUaVal;
CpuMemoryUsage(NetID := NetID); // ReadMemoryUsage
PlcDiagState[1](
    LineName := GVL_const.LineName,
    MachineName := GVL_const.MachineName,
    StateName := GVL_const.PlcCpuMemUsage,
    TimeStamp := GVL_SW.Unix_TimeStamp,
    Value := UINT_TO_INT(CpuMemoryUsage.MemUsage)); // GenericState

// PAGE PLC CPU usage ---
PlcCpuCore2UsageStruct := PlcDiagState[2].OpcUaVal;
CpuUsageEx_Core2(bExecute := tonRecycle50ms.Q, tTimeout := T#5S, sNetId := NetID, nCpuId := 2); // TC_CPuUsageEx
PlcDiagState[2](
    LineName := GVL_const.LineName,
    MachineName := GVL_const.MachineName,
    StateName := GVL_const.PlcCpuCore2Usage,
    TimeStamp := GVL_SW.Unix_TimeStamp,
    Value := UDINT_TO_INT(CpuUsageEx_Core2.nUsage),
    Enable := GVL_Visu.LineRunning AND tonRecyclePublishMqtt.Q); // GenericState
PlcCpuCore3UsageStruct := PlcDiagState[3].OpcUaVal;
CpuUsageEx_Core3(bExecute := tonRecycle50ms.Q, tTimeout := T#5S, sNetId := NetID, nCpuId := 3); // TC_CPuUsageEx
PlcDiagState[3](
    LineName := GVL_const.LineName,
    MachineName := GVL_const.MachineName,
    StateName := GVL_const.PlcCpuCore3Usage,
    TimeStamp := GVL_SW.Unix_TimeStamp,
    Value := UDINT_TO_INT(CpuUsageEx_Core3.nUsage),
    Enable := GVL_Visu.LineRunning AND tonRecyclePublishMqtt.Q); // GenericState

// PAGE PLC CPU latency
CpuLatencyEx_Core2(bExecute := tonRecycle50ms.Q, tTimeout := T#5S, sNetId := NetID, nCpuId := 2); // TC_SysLatencyEx
PlcDiagState[4](
    LineName := GVL_const.LineName,
    MachineName := GVL_const.MachineName,
    StateName := GVL_const.PlcCpuCore2Jitter,
    TimeStamp := GVL_SW.Unix_TimeStamp,
    Value := UDINT_TO_INT(CpuLatencyEx_Core2.nActual),
    Enable := GVL_Visu.LineRunning AND tonRecyclePublishMqtt.Q); // GenericState
PlcCpuCore2JitterStruct := PlcDiagState[4].OpcUaVal;
PlcCpuCore3JitterStruct := PlcDiagState[5].OpcUaVal;
CpuLatencyEx_Core3(bExecute := tonRecycle50ms.Q, tTimeout := T#5S, sNetId := NetID, nCpuId := 3); // TC_SysLatencyEx
PlcDiagState[5](
    LineName := GVL_const.LineName,
    MachineName := GVL_const.MachineName,
    StateName := GVL_const.PlcCpuCore3Jitter,
    TimeStamp := GVL_SW.Unix_TimeStamp,
    Value := UDINT_TO_INT(CpuLatencyEx_Core3.nActual),
    Enable := GVL_Visu.LineRunning AND tonRecyclePublishMqtt.Q); // GenericState
// GVL_Visu.LineRunning AND tonRecyclePublishMqtt.Q: input not connected

END_PROGRAM

// ---- POUs/FB/Generic/ReadMemoryUsage.TcPOU
FUNCTION_BLOCK ReadMemoryUsage

VAR_INPUT
	NetID				: 	STRING;
END_VAR

VAR
	  
    eStateMemTotal      : BYTE;            	  // index for state machine Total Memory allocated 
	eStateMemAvail      : BYTE;               // index for state machine Memory Available   
    bStartMemTotal      : BOOL := TRUE;       // flag to trigger (re)start of statemachine
	bStartMemAvail      : BOOL := TRUE;       // flag to trigger (re)start of statemachine
    nDataMemTotal       : ULINT;              // data storage for Total Memory 
    nDataMemAvail       : ULINT;              // data storage for Memory Avaiable
    stMDP_AddrMemTotal  : ST_MDP_Addr;        // structure for MDP addresses  
    stMDP_AddrMemAvail  : ST_MDP_Addr;        // structure for MDP addresses
	
    // FB instances
    fbReadMDPElementMemTotal    : FB_MDP_ReadElement; // instance of FB for reading MDP element 
	fbReadMDPElementMemAvail    : FB_MDP_ReadElement; // instance of FB for reading MDP element 

    // execution results
    bErrorMemTotal              : BOOL;               // error flag (indicator: error occured)
    nErrIDMemTotal              : UDINT;              // last error ID
    nMemTotalAllocated          : ULINT;              // total memory allocated [bytes] 
	
	// execution results
    bErrorMemAvail              : BOOL;               // error flag (indicator: error occured)
    nErrIDMemAvail              : UDINT;              // last error ID
    nMemAvailable               : ULINT;              // memory available [bytes]

END_VAR

VAR_OUTPUT
	MemUsage					: UINT;			  	  // current memory usage [%]
END_VAR

(*
This FB reads out current values of total memory and 
memory available on the target system.
It works properly on Beckhoff HW.
*)

CASE eStateMemTotal OF
    0: 
        IF bStartMemTotal THEN
            bStartMemTotal := FALSE;
            eStateMemTotal := 1; 							//** initiate first state
        END_IF

    1:    
        stMDP_AddrMemTotal.nArea    := INT_TO_BYTE(eMDP_Area_ConfigArea); 	// set area address to "Config Area"
        stMDP_AddrMemTotal.nTableId := 1;              						// table ID in module for "cpu properties"
        stMDP_AddrMemTotal.nSubIdx  := 6;              						// subindex in table ID for "CPU usage"    
																			// 06=program memory allocated (>4GB RAM)
									            							// 07=program memory available (>4GB RAM)                 
        
        fbReadMDPElementMemTotal(
            bExecute    := TRUE,               	  // Flag: trigger execution of FB
             
			eModuleType := eMDP_ModT_Memory, 	  // desired module type = Memory       
            stMDP_Addr  := stMDP_AddrMemTotal,    // MDP address structure. Dynamic module ID added internally. 
            iModIdx     := 0,                     // instance of desired module type (0 = first instance) 
            pDstBuf     := ADR(nDataMemTotal),    // buffer for storing data
            cbDstBufLen := SIZEOF(nDataMemTotal), // length of buffer
            sAmsNetId   := NetID,          
            );                                    // Note: fbReadMDPElement.tTimeOut must be > cycle time!

        eStateMemTotal := 2;  					  // next state: process FB
            
    2:                
        fbReadMDPElementMemTotal(bExecute := FALSE);    // Flag: Get execution state of FB 
                                               	  		//** Note: fbReadMDPElement.tTimeOut must be > cycle time!

        IF NOT fbReadMDPElementMemTotal.bBusy THEN     
            IF fbReadMDPElementMemTotal.bError THEN    
                bErrorMemTotal    := TRUE;             					// set error flag
                nErrIDMemTotal    := fbReadMDPElementMemTotal.nErrID; 	// store error id (16#ECA60105 = BIOS or HW does 
                                               							// not support this data (here: mainboard data))
                eStateMemTotal    := 0;				   					// finish state machine
            ELSE                               							
                bErrorMemTotal    := FALSE;            					
                nMemTotalAllocated := nDataMemTotal;            		// store in dedicated variable
                eStateMemTotal    := 1; 			   					// next state 
            END_IF
        END_IF
    
END_CASE 


CASE eStateMemAvail OF
    0: 
        IF bStartMemAvail THEN
            bStartMemAvail := FALSE;
            eStateMemAvail := 1; //** initiate first state
        END_IF

    1:    
        stMDP_AddrMemAvail.nArea    := INT_TO_BYTE(eMDP_Area_ConfigArea); //** set area address to "Config Area"
        stMDP_AddrMemAvail.nTableId := 1;              //** table ID in module for "cpu properties"
        stMDP_AddrMemAvail.nSubIdx  := 7;              //** subindex in table ID for "CPU usage"                     
        
        fbReadMDPElementMemAvail(
            bExecute    := TRUE,               			// Flag: trigger execution of FB
            //eModuleType := eMDP_ModT_CPU,      		//** desired module type = CPU 
			eModuleType := eMDP_ModT_Memory,        
            stMDP_Addr  := stMDP_AddrMemAvail,         	// MDP address structure. Dynamic module ID added internally. 
            iModIdx     := 0,                  			//** instance of desired module type (0 = first instance) 
            pDstBuf     := ADR(nDataMemAvail),         	// buffer for storing data
            cbDstBufLen := SIZEOF(nDataMemAvail),      	// length of buffer
            sAmsNetId   := NetID,          				// AMS Net ID
            );                                 			//** Note: fbReadMDPElement.tTimeOut must be > cycle time!

        eStateMemAvail := 2;  					   	   	//** next state: process FB
            
    2:                									//** process FB: request CPU data
        fbReadMDPElementMemAvail(bExecute := FALSE);   	// Flag: Get execution state of FB 
                                               			//** Note: fbReadMDPElement.tTimeOut must be > cycle time!

        IF NOT fbReadMDPElementMemAvail.bBusy THEN     						// FB executed?
            IF fbReadMDPElementMemAvail.bError THEN    						// Error?
                bErrorMemAvail    := TRUE;             						// set error flag
                nErrIDMemAvail    := fbReadMDPElementMemAvail.nErrID; 		// store error id (16#ECA60105 = BIOS or HW does 
                                               								// not support this data (here: mainboard data))
                eStateMemAvail    := 0;				   						// finish state machine
            ELSE                               								// set parameters for next steps
                bErrorMemAvail    := FALSE;            						// turn off error flag
                nMemAvailable := nDataMemAvail;            					//** store CPU usage in dedicated variable
                eStateMemAvail    := 1; 			   						//** next state 
            END_IF
        END_IF
    
END_CASE 

// calculate current memory usage as difference between total memory - available memory
IF nMemTotalAllocated <>0 THEN
	MemUsage := REAL_TO_UINT(100 * ULINT_TO_REAL(nMemTotalAllocated - nMemAvailable)/ULINT_TO_REAL(nMemTotalAllocated));
END_IF

END_FUNCTION_BLOCK

// ---- POUs/PRG_10ms/PRG_11_AirFlowAnalytics.TcPOU
PROGRAM PRG_11_AirFlowAnalytics
VAR
	AirFlowRateSensor: GenericSensor;
	AirPressureSensor: GenericSensor;
	AirTemperatureSensor: GenericSensor;
	
	{attribute 'OPC.UA.DA' := '0'}
	{attribute 'OPC.UA.DA.Access' := '1'}			// read only
	{attribute 'OPC.UA.DA.StructuredType' := '1'}
	AirFlowRateSensorStruct						: SingleSensor_DataModel;
	
	{attribute 'OPC.UA.DA' := '0'}
	{attribute 'OPC.UA.DA.Access' := '1'}			// read only
	{attribute 'OPC.UA.DA.StructuredType' := '1'}
	AirPressureSensorStruct						: SingleSensor_DataModel;
	
	{attribute 'OPC.UA.DA' := '0'}
	{attribute 'OPC.UA.DA.Access' := '1'}			// read only
	{attribute 'OPC.UA.DA.StructuredType' := '1'}
	AirTemperatureSensorSensorStruct			: SingleSensor_DataModel;
END_VAR

AirFlowRateSensor(
    LineName := GVL_const.LineName,
    MachineName := GVL_const.MachineName,
    SensorName := GVL_const.AirFlowSensor,
    TimeStamp := GVL_SW.Unix_TimeStamp,
    Value := GVL_Visu.AirFlowRate,
    Enable := GVL_Visu.LineRunning); // GenericSensor
AirFlowRateSensorStruct := AirFlowRateSensor.OpcUaVal;
AirPressureSensor(
    LineName := GVL_const.LineName,
    MachineName := GVL_const.MachineName,
    SensorName := GVL_const.AirPresSensor,
    TimeStamp := GVL_SW.Unix_TimeStamp,
    Value := GVL_Visu.AirPressure,
    Enable := GVL_Visu.LineRunning); // GenericSensor
AirPressureSensorStruct := AirPressureSensor.OpcUaVal;
AirTemperatureSensor(
    LineName := GVL_const.LineName,
    MachineName := GVL_const.MachineName,
    SensorName := GVL_const.AirTempSensor,
    TimeStamp := GVL_SW.Unix_TimeStamp,
    Value := GVL_Visu.AirTemperature,
    Enable := GVL_Visu.LineRunning); // GenericSensor
AirTemperatureSensorSensorStruct := AirTemperatureSensor.OpcUaVal;
// GVL_SW.AirVolumetricFlowRate: input not connected
// GVL_SW.AirPressure: input not connected
// GVL_SW.AirTemperature: input not connected

END_PROGRAM

// ---- POUs/FB/OPC_UA/GenericSensor.TcPOU
FUNCTION_BLOCK GenericSensor
VAR_INPUT
	LineName	: STRING(40);
	MachineName : STRING(40);
	SensorName	: STRING(40);
	TimeStamp	: ULINT;
	Value		: REAL;	 
	Enable		: BOOL; //enable sensor evaluation
END_VAR
VAR_OUTPUT
	OpcUaVal		: SingleSensor_DataModel;
END_VAR
VAR
	SetParameter : BOOL := TRUE;	
	
	stValues		: SingleSensor_DataModel;	
	
	// safety watchdog
	tonWatchdog : TON;
END_VAR

(*
This FB evaluates analog value and creates output struct for OPC UA
*) 

IF Enable THEN
	
	IF SetParameter THEN
		SetParameter := FALSE;
		// constant entry
		stValues.LineName := LineName;
		stValues.MachineName := MachineName;
		stValues.SensorName := SensorName;
	END_IF
	
	stValues.timeStamp := TimeStamp;
	stValues.SensorValue := Value;
		
	OpcUaVal := stValues;
ELSE
	;
END_IF;

END_FUNCTION_BLOCK

// ---- POUs/PRG_10ms/PRG_10_TempHumidAnalytics.TcPOU
PROGRAM PRG_10_TempHumidAnalytics
VAR
	TempSensor								: GenericSensor;
	HumiditySensor							: GenericSensor;
	
	{attribute 'OPC.UA.DA' := '1'}					// enable/disable to OPC UA
	{attribute 'OPC.UA.DA.Access' := '1'}			// read only
	{attribute 'OPC.UA.DA.StructuredType' := '1'}	// define variable as STRUCT for OPC UA
	TempSensorStruct						: SingleSensor_DataModel;
	
	{attribute 'OPC.UA.DA' := '1'}					// enable/disable to OPC UA
	{attribute 'OPC.UA.DA.Access' := '1'}			// read only
	{attribute 'OPC.UA.DA.StructuredType' := '1'}	// define variable as STRUCT for OPC UA
	HumiditySensorStruct					: SingleSensor_DataModel;
END_VAR

TempSensorStruct := TempSensor.OpcUaVal;
TempSensor(
    LineName := GVL_const.LineName,
    MachineName := GVL_const.MachineName,
    SensorName := GVL_const.AmbientTempSensor,
    TimeStamp := GVL_SW.Unix_TimeStamp,
    Value := GVL_Visu.AmbientTemperature,
    Enable := GVL_Visu.LineRunning); // GenericSensor
HumiditySensorStruct := HumiditySensor.OpcUaVal;
HumiditySensor(
    LineName := GVL_const.LineName,
    MachineName := GVL_const.MachineName,
    SensorName := GVL_const.AmbientHumiditySensor,
    TimeStamp := GVL_SW.Unix_TimeStamp,
    Value := GVL_Visu.AmbientHumidity,
    Enable := GVL_Visu.LineRunning); // GenericSensor
// GVL_SW.AmbientTempSensor: input not connected
// GVL_SW.AmbientHumiditySensor: input not connected

END_PROGRAM

// ---- POUs/PRG_10ms/PRG_12_OilContaminationAnalytics.TcPOU
PROGRAM PRG_12_OilContaminationAnalytics
VAR
	OilDiffPressSensor: GenericSensor;
	
	{attribute 'OPC.UA.DA' := '1'}
	{attribute 'OPC.UA.DA.Access' := '1'}			// read only
	{attribute 'OPC.UA.DA.StructuredType' := '1'}
	OilDiffPressSensorStruct			: SingleSensor_DataModel;
END_VAR

OilDiffPressSensorStruct := OilDiffPressSensor.OpcUaVal;
OilDiffPressSensor(
    LineName := GVL_const.LineName,
    MachineName := GVL_const.MachineName,
    SensorName := GVL_const.DiffPressSensor1,
    TimeStamp := GVL_SW.Unix_TimeStamp,
    Value := GVL_Visu.OilDiffPressure,
    Enable := GVL_Visu.LineRunning); // GenericSensor
// GVL_SW.DiffPressSensor: input not connected

END_PROGRAM

// ---- POUs/PRG_1ms/Main_T1ms.TcPOU
PROGRAM Main_T1ms
VAR
			 
END_VAR

// time stamp generation
TimeStamp();

END_PROGRAM

// ---- POUs/EL3443/EL3443_DPM/FB_EL3443_DPM.TcPOU
(*  This function block calls up the variant values supplied by the EL3443 terminal. The multiplexer channels of the terminal are queried by the use of selectors.
    Due to the multiplexing of the values in the variant values, reading the terminal information requires several PLC cycles.
    In contrast, values that can be retrieved via the process image are output cyclically. 
    
    To use the function block:
    ▪ the predefined PDO assignment "DPM" (DPM: Distributed Power Measurement) must be selected for the terminal under "Process data".
    
    ▪ Then the PLC data type (structure from the process data, MDP5001_341_93A85FAB) must be activated in the "PLC" tab of the terminal.
    
    ▪ After creating the data type, the PLC project must be rebuilt.
    
    ▪ Finally, the terminal must be linked to the function block on the "PLC" tab*)

{attribute 'no-analysis'}  
{attribute 'hide_all_locals'}         
FUNCTION_BLOCK FB_EL3443_DPM
VAR_INPUT
    bEnable : BOOL; //Enables the Variant values to be queried using the multiplexer functions of the block
	
    stEL3443_IO : MDP5001_341_93A85FAB; //External data type that can be generated within the terminal on the PLC tab
				// new MDP5001_341_93A85FAB
				// old MDP5001_341_93A85FAB
END_VAR

VAR_OUTPUT
    stStatusTotal 	 : ST_EL3443_DPM_StatusTotal; //General cyclical process data
    stStatusPhase_L1 : ST_EL3443_DPM_StatusLx; //Phase L1 specific cyclical process data 
    stStatusPhase_L2 : ST_EL3443_DPM_StatusLx; //Phase L2 specific cyclical process data
    stStatusPhase_L3 : ST_EL3443_DPM_StatusLx; //Phase L3 specific cyclical process data
    stVariantValues  : ST_EL3443_DPM_VariantValues; //Variant Values (non-cyclical values). Due to the multiplexing of the values in the Variant Values, the reading of the terminal information requires several PLC cycles.
    
    pDpmData : POINTER TO ARRAY[1..20] OF UDINT;
    
    bError : BOOL; //Becomes TRUE as soon as an error situation occurs.
END_VAR

VAR
    {attribute 'no_copy'}
    astEL3443MuxReal_Ch1: ARRAY [0..nARRAYSIZEMUXREAL] OF ST_EL3443_DPM_MUX_REAL; //Structure for the (Real) Multiplexer Channel 1 contains the selector and a reference to the corresponding memory location
    {attribute 'no_copy'}
    astEL3443MuxReal_Ch2: ARRAY [0..nARRAYSIZEMUXREAL] OF ST_EL3443_DPM_MUX_REAL; //Structure for the (Real) Multiplexer Channel 2 contains the selector and a reference to the corresponding memory location
    {attribute 'no_copy'}
    astEL3443MuxReal_Ch3: ARRAY [0..nARRAYSIZEMUXREAL] OF ST_EL3443_DPM_MUX_REAL; //Structure for the (Real) Multiplexer Channel 3 contains the selector and a reference to the corresponding memory location
    {attribute 'no_copy'}
    stEL3443MuxUlint_Ch4: ARRAY [0..nARRAYSIZEMUXULINT] OF ST_EL3443_DPM_MUX_ULINT; //Structure for the (ULINT/LINT) multiplexer channel 4 contains the selector and a pointer to the corresponding memory location
    
    {attribute 'no_copy'}
    bInit : BOOL; //Flag to indicate the initialised state of the function block
    nMuxRealState : INT := 0; //Position der Multplexer-Abfragen (Channel 1-3 (REAL))
    nCounterNotRepliedMuxReal : INT; //Number of cycles in which the multiplexer has not responded
    nMuxUlintState : INT := 0; //Position der Multplexer-Abfragen (Channel 4 (ULINT))
    nCounterNotRepliedMuxUlint : INT; //Number of cycles in which the multiplexer has not responded
    
    {attribute 'no_copy'}
    nNumberOfSelectorsCh1 : UINT; //number of selectors in channel 1
    {attribute 'no_copy'}
    nNumberOfSelectorsCh2 : UINT; //number of selectors in channel 2
    {attribute 'no_copy'}
    nNumberOfSelectorsCh3 : UINT; //number of selectors in channel 3
    {attribute 'no_copy'}
    nNumberOfSelectorsCh4 : UINT; //number of selectors in channel 4      
END_VAR

VAR CONSTANT
    nARRAYSIZEMUXREAL : INT := 122; //Array size of the REAL multiplexer channel
    nARRAYSIZEMUXULINT : INT := 74; //Array size of the ULINT multiplexer channel
    nERROR_NOT_REPLIED : INT := 10; //Maximum number of cycles the multiplexer may use before the error output is set 
END_VAR

//The output bError is set if the block is enabled and one of the multiplexer channels does not respond
bError := bEnable AND (nCounterNotRepliedMuxUlint >= nERROR_NOT_REPLIED OR nCounterNotRepliedMuxReal >= nERROR_NOT_REPLIED) ;

IF bEnable THEN
      
    IF NOT bInit THEN
        bInit := TRUE;
        Initialize();
    END_IF
    
    //===================================================================================================================================
    // Multiplexer channels 1-3 (REAL)
    
    //comparison of the transmitting and receiving selectors 
    IF astEL3443MuxReal_Ch1[nMuxRealState].nSelector = stEL3443_IO.MDP5001_341_Input.MDP5001_341_Total_Variant_Value_In_Index_1_REAL AND
       astEL3443MuxReal_Ch2[nMuxRealState].nSelector = stEL3443_IO.MDP5001_341_Input.MDP5001_341_Total_Variant_Value_In_Index_2_REAL AND 
       astEL3443MuxReal_Ch3[nMuxRealState].nSelector = stEL3443_IO.MDP5001_341_Input.MDP5001_341_Total_Variant_Value_In_Index_3_REAL THEN
        
    
        //assignment of the received values to the referenced references
        IF __ISVALIDREF(astEL3443MuxReal_Ch1[nMuxRealState].fValueRef) THEN
            astEL3443MuxReal_Ch1[nMuxRealState].fValueRef := stEL3443_IO.MDP5001_341_Input.MDP5001_341_Total_Variant_Value_In_Value_1_REAL;
        END_IF
        IF __ISVALIDREF(astEL3443MuxReal_Ch2[nMuxRealState].fValueRef) THEN
            astEL3443MuxReal_Ch2[nMuxRealState].fValueRef := stEL3443_IO.MDP5001_341_Input.MDP5001_341_Total_Variant_Value_In_Value_2_REAL;
        END_IF
        IF __ISVALIDREF(astEL3443MuxReal_Ch3[nMuxRealState].fValueRef) THEN
            astEL3443MuxReal_Ch3[nMuxRealState].fValueRef := stEL3443_IO.MDP5001_341_Input.MDP5001_341_Total_Variant_Value_In_Value_3_REAL;
        END_IF
       
       //selection of the new selector group
       nMuxRealState := nMuxRealState + 1;
     
       IF nMuxRealState > nARRAYSIZEMUXREAL THEN
         nMuxRealState := 0;  
       END_IF
       
       nCounterNotRepliedMuxReal := 0;
    ELSIF
        stEL3443_IO.MDP5001_341_Input.MDP5001_341_Total_Variant_Value_In_Index_1_REAL = E_EL3443_DPM_Phase.Error_INDEX_Not_Valid OR    
        stEL3443_IO.MDP5001_341_Input.MDP5001_341_Total_Variant_Value_In_Index_2_REAL = E_EL3443_DPM_Phase.Error_INDEX_Not_Valid OR 
        stEL3443_IO.MDP5001_341_Input.MDP5001_341_Total_Variant_Value_In_Index_3_REAL = E_EL3443_DPM_Phase.Error_INDEX_Not_Valid THEN
    
        nCounterNotRepliedMuxReal := MIN(nCounterNotRepliedMuxReal + 1,nERROR_NOT_REPLIED);
    ELSE
        nCounterNotRepliedMuxReal := MIN(nCounterNotRepliedMuxReal + 1,nERROR_NOT_REPLIED); 
    END_IF
       
    // transfer of the selectors to the process image 
    stEL3443_IO.MDP5001_341_Output.MDP5001_341_Total_Variant_Value_Out_Index_1_REAL := astEL3443MuxReal_Ch1[nMuxRealState].nSelector;
    stEL3443_IO.MDP5001_341_Output.MDP5001_341_Total_Variant_Value_Out_Index_2_REAL := astEL3443MuxReal_Ch2[nMuxRealState].nSelector;
    stEL3443_IO.MDP5001_341_Output.MDP5001_341_Total_Variant_Value_Out_Index_3_REAL := astEL3443MuxReal_Ch3[nMuxRealState].nSelector;
    
    //===================================================================================================================================
    // Multiplexer channels 4 (ULINT)
    
    //comparison of the transmitting and receiving selector
    IF stEL3443MuxUlint_Ch4[nMuxUlintState].nSelector = stEL3443_IO.MDP5001_341_Input.MDP5001_341_Total_Variant_Value_In_Index_4_ULINT THEN
        
        //assigns the received values to the assigned pointer address.
        IF stEL3443MuxUlint_Ch4[nMuxUlintState].nValueRef <> 0 THEN
            stEL3443MuxUlint_Ch4[nMuxUlintState].nValueRef^ := stEL3443_IO.MDP5001_341_Input.MDP5001_341_Total_Variant_Value_In_Value_4_ULINT;
        END_IF
        
    //selection of the new selector group
       nMuxUlintState := nMuxUlintState + 1;
     
       IF nMuxUlintState > nARRAYSIZEMUXULINT THEN
         nMuxUlintState := 0;  
       END_IF
       
       nCounterNotRepliedMuxUlint := 0;
    ELSIF stEL3443_IO.MDP5001_341_Input.MDP5001_341_Total_Variant_Value_In_Index_4_ULINT = E_EL3443_DPM_Phase.Error_INDEX_Not_Valid THEN
    
        nCounterNotRepliedMuxUlint := MIN(nCounterNotRepliedMuxUlint + 1, nERROR_NOT_REPLIED);
    ELSE
        nCounterNotRepliedMuxUlint := MIN(nCounterNotRepliedMuxUlint + 1, nERROR_NOT_REPLIED);  
    END_IF
    
    // transfer of the selectors to the process image
    stEL3443_IO.MDP5001_341_Output.MDP5001_341_Total_Variant_Value_Out_Index_4_ULINT := stEL3443MuxUlint_Ch4[nMuxUlintState].nSelector;
END_IF

//===================================================================================================================================
// Update the cyclic outputs

// Set pointer address to transmit DPM communication information
pDpmData := ADR(stEL3443_IO.MDP5001_341_Input.MDP5001_341_DPM_Data_Data_1);

// Transfer of process data to PLC common data types. Status total.
stStatusTotal.bStatus_System_State :=                       stEL3443_IO.MDP5001_341_Input.MDP5001_341_Total_Status_System_State;
stStatusTotal.bStatus_Grid_Direction :=                     stEL3443_IO.MDP5001_341_Input.MDP5001_341_Total_Status_Grid_Direction;
stStatusTotal.bStatus_Frequency_Guard_Warning :=            stEL3443_IO.MDP5001_341_Input.MDP5001_341_Total_Status_Frequency_Guard_Warning;
stStatusTotal.bStatus_Frequency_Guard_Error :=              stEL3443_IO.MDP5001_341_Input.MDP5001_341_Total_Status_Frequency_Guard_Error;
stStatusTotal.bStatus_Neutral_Current_Guard_Warning :=      stEL3443_IO.MDP5001_341_Input.MDP5001_341_Total_Status_Neutral_Current_Guard_Warning;
stStatusTotal.bStatus_Neutral_Current_Guard_Error :=        stEL3443_IO.MDP5001_341_Input.MDP5001_341_Total_Status_Neutral_Current_Guard_Error;
stStatusTotal.bStatus_Active_Power_Guard_Warning :=         stEL3443_IO.MDP5001_341_Input.MDP5001_341_Total_Status_Active_Power_Guard_Warning;    
stStatusTotal.bStatus_Active_Power_Guard_Error :=           stEL3443_IO.MDP5001_341_Input.MDP5001_341_Total_Status_Active_Power_Guard_Error;
stStatusTotal.bStatus_Apparent_Power_Guard_Warning :=       stEL3443_IO.MDP5001_341_Input.MDP5001_341_Total_Status_Apparent_Power_Guard_Warning;
stStatusTotal.bStatus_Apparent_Power_Guard_Error :=         stEL3443_IO.MDP5001_341_Input.MDP5001_341_Total_Status_Apparent_Power_Guard_Error; 
stStatusTotal.bStatus_Power_Quality_Guard_Warning :=        stEL3443_IO.MDP5001_341_Input.MDP5001_341_Total_Status_Power_Quality_Guard_Warning; 
stStatusTotal.bStatus_Power_Quality_Guard_Error :=          stEL3443_IO.MDP5001_341_Input.MDP5001_341_Total_Status_Power_Quality_Guard_Error; 
stStatusTotal.bStatus_TxPDO_State :=                        stEL3443_IO.MDP5001_341_Input.MDP5001_341_Total_Status_TxPDO_State; 
stStatusTotal.bStatus_TxPDO_Toggle :=                       stEL3443_IO.MDP5001_341_Input.MDP5001_341_Total_Status_TxPDO_Toggle; 
stStatusTotal.fStatus_Power_Quality_Factor :=               stEL3443_IO.MDP5001_341_Input.MDP5001_341_Total_Status_Power_Quality_Factor; 

